LIN {X 0,Y 407.293,Z 572.545,A -85,B 0,C 180,E1 -11318.769,E2 -11318.769} C_VEL
LIN {X 0,Y 407.261,Z 605.136,A -85,B 0,C 180,E1 -11319.46,E2 -11319.46} C_VEL
LIN {X 0,Y 407.213,Z 619.891,A -85,B 0,C 180,E1 -11319.972,E2 -11319.972} C_VEL
LIN {X 0,Y 406.821,Z 633.745,A -85,B 0,C 180,E1 -11320.641,E2 -11320.641} C_VEL
LIN {X 0,Y 406.274,Z 646.742,A -85,B 0,C 180,E1 -11321.466,E2 -11321.466} C_VEL
LIN {X 0,Y 405.576,Z 659.147,A -85,B 0,C 180,E1 -11322.444,E2 -11322.444} C_VEL
LIN {X 0,Y 404.643,Z 671.423,A -85,B 0,C 180,E1 -11323.636,E2 -11323.636} C_VEL
LIN {X 0,Y 403.725,Z 681.881,A -85,B 0,C 180,E1 -11324.863,E2 -11324.863} C_VEL
LIN {X 0,Y 402.584,Z 692.537,A -85,B 0,C 180,E1 -11326.368,E2 -11326.368} C_VEL
LIN {X 0,Y 401.584,Z 701.412,A -85,B 0,C 180,E1 -11327.877,E2 -11327.877} C_VEL
LIN {X 0,Y 400.622,Z 709.855,A -85,B 0,C 180,E1 -11329.61,E2 -11329.61} C_VEL
LIN {X 0,Y 399.757,Z 716.985,A -85,B 0,C 180,E1 -11331.405,E2 -11331.405} C_VEL
LIN {X 0,Y 398.956,Z 721.911,A -85,B 0,C 180,E1 -11332.916,E2 -11332.916} C_VEL
LIN {X 0,Y 398.421,Z 727.092,A -85,B 0,C 180,E1 -11334.94,E2 -11334.94} C_VEL
LIN {X 0,Y 397.856,Z 730.905,A -85,B 0,C 180,E1 -11336.962,E2 -11336.962} C_VEL
LIN {X 0,Y 397.512,Z 733.428,A -85,B 0,C 180,E1 -11338.987,E2 -11338.987} C_VEL
LIN {X 0,Y 397.294,Z 734.718,A -85,B 0,C 180,E1 -11341.013,E2 -11341.013} C_VEL
LIN {X 0,Y 397.207,Z 734.793,A -85,B 0,C 180,E1 -11343.042,E2 -11343.042} C_VEL
LIN {X 0,Y 397.117,Z 733.67,A -85,B 0,C 180,E1 -11345.076,E2 -11345.076} C_VEL
LIN {X 0,Y 397.307,Z 731.92,A -85,B 0,C 180,E1 -11346.634,E2 -11346.634} C_VEL
LIN {X 0,Y 397.376,Z 729.649,A -85,B 0,C 180,E1 -11348.133,E2 -11348.133} C_VEL
LIN {X 0,Y 397.643,Z 725.336,A -85,B 0,C 180,E1 -11350.18,E2 -11350.18} C_VEL
LIN {X 0,Y 397.959,Z 719.588,A -85,B 0,C 180,E1 -11352.234,E2 -11352.234} C_VEL
LIN {X 0,Y 398.554,Z 712.207,A -85,B 0,C 180,E1 -11354.292,E2 -11354.292} C_VEL
LIN {X 0,Y 399.245,Z 704.203,A -85,B 0,C 180,E1 -11356.096,E2 -11356.096} C_VEL
LIN {X 0,Y 400.049,Z 694.472,A -85,B 0,C 180,E1 -11357.904,E2 -11357.904} C_VEL
LIN {X 0,Y 400.824,Z 684.417,A -85,B 0,C 180,E1 -11359.459,E2 -11359.459} C_VEL
LIN {X 0,Y 401.695,Z 673.415,A -85,B 0,C 180,E1 -11360.884,E2 -11360.884} C_VEL
LIN {X 0,Y 402.54,Z 661.884,A -85,B 0,C 180,E1 -11362.136,E2 -11362.136} C_VEL
LIN {X 0,Y 403.272,Z 649.96,A -85,B 0,C 180,E1 -11363.222,E2 -11363.222} C_VEL
LIN {X 0,Y 404.01,Z 635.883,A -85,B 0,C 180,E1 -11364.265,E2 -11364.265} C_VEL
LIN {X 0,Y 404.662,Z 621.146,A -85,B 0,C 180,E1 -11365.12,E2 -11365.12} C_VEL
LIN {X 0,Y 405.075,Z 605.669,A -85,B 0,C 180,E1 -11365.793,E2 -11365.793} C_VEL
LIN {X 0,Y 405.206,Z 590.616,A -85,B 0,C 180,E1 -11366.244,E2 -11366.244} C_VEL
LIN {X 0,Y 405.225,Z 572.67,A -85,B 0,C 180,E1 -11366.637,E2 -11366.637} C_VEL
LIN {X 0,Y 397.184,Z 551.01,A -85,B 0,C 180,E1 -11367.501,E2 -11367.501} C_VEL
LIN {X 0,Y 397.08,Z 551.019,A -85,B 0,C 180,E1 -11370.882,E2 -11370.882} C_VEL
LIN {X 0,Y 397.126,Z 551.016,A -85,B 0,C 180,E1 -11374.493,E2 -11374.493} C_VEL
LIN {X 0,Y 397.103,Z 551.022,A -85,B 0,C 180,E1 -11378.274,E2 -11378.274} C_VEL
LIN {X 0,Y 397.089,Z 551.018,A -85,B 0,C 180,E1 -11380.908,E2 -11380.908} C_VEL
LIN {X 0,Y 397.101,Z 551.017,A -85,B 0,C 180,E1 -11383.648,E2 -11383.648} C_VEL
LIN {X 0,Y 397.102,Z 551.021,A -85,B 0,C 180,E1 -11386.52,E2 -11386.52} C_VEL
LIN {X 0,Y 397.115,Z 551.022,A -85,B 0,C 180,E1 -11390.422,E2 -11390.422} C_VEL
LIN {X 0,Y 397.108,Z 551.02,A -85,B 0,C 180,E1 -11394.265,E2 -11394.265} C_VEL
LIN {X 0,Y 397.114,Z 551.019,A -85,B 0,C 180,E1 -11396.726,E2 -11396.726} C_VEL
LIN {X 0,Y 397.124,Z 551.017,A -85,B 0,C 180,E1 -11400.295,E2 -11400.295} C_VEL
LIN {X 0,Y 397.193,Z 551.012,A -85,B 0,C 180,E1 -11402.609,E2 -11402.609} C_VEL
LIN {X 0,Y 397.132,Z 551.013,A -85,B 0,C 180,E1 -11405.981,E2 -11405.981} C_VEL
LIN {X 0,Y 397.137,Z 551.011,A -85,B 0,C 180,E1 -11409.704,E2 -11409.704} C_VEL
LIN {X 0,Y 397.18,Z 551.014,A -85,B 0,C 180,E1 -11412.844,E2 -11412.844} C_VEL
LIN {X 0,Y 397.225,Z 551.005,A -85,B 0,C 180,E1 -11416.678,E2 -11416.678} C_VEL
LIN {X 0,Y 397.217,Z 551.002,A -85,B 0,C 180,E1 -11419.808,E2 -11419.808} C_VEL
LIN {X 0,Y 397.362,Z 550.989,A -85,B 0,C 180,E1 -11422.888,E2 -11422.888} C_VEL
LIN {X 0,Y 397.254,Z 551.003,A -85,B 0,C 180,E1 -11424.925,E2 -11424.925} C_VEL
LIN {X 0,Y 397.45,Z 550.973,A -85,B 0,C 180,E1 -11427.973,E2 -11427.973} C_VEL
LIN {X 0,Y 397.579,Z 550.957,A -85,B 0,C 180,E1 -11429.999,E2 -11429.999} C_VEL
LIN {X 0,Y 397.38,Z 550.987,A -85,B 0,C 180,E1 -11433.041,E2 -11433.041} C_VEL
LIN {X 0,Y 397.357,Z 550.989,A -85,B 0,C 180,E1 -11437.111,E2 -11437.111} C_VEL
LIN {X 0,Y 397.22,Z 551.001,A -85,B 0,C 180,E1 -11440.19,E2 -11440.19} C_VEL
LIN {X 0,Y 397.223,Z 551.008,A -85,B 0,C 180,E1 -11443.32,E2 -11443.32} C_VEL
LIN {X 0,Y 397.165,Z 551.009,A -85,B 0,C 180,E1 -11446.89,E2 -11446.89} C_VEL
LIN {X 0,Y 396.521,Z 551.096,A -85,B 0,C 180,E1 -11447.737,E2 -11447.737} C_VEL
LIN {X 0,Y 393.659,Z 551.454,A -85,B 0,C 180,E1 -11449.111,E2 -11449.111} C_VEL
LIN {X 0,Y 391.208,Z 551.757,A -85,B 0,C 180,E1 -11450.222,E2 -11450.222} C_VEL
LIN {X 0,Y 390.138,Z 551.886,A -85,B 0,C 180,E1 -11451.081,E2 -11451.081} C_VEL
LIN {X 0,Y 390.042,Z 551.896,A -85,B 0,C 180,E1 -11451.373,E2 -11451.373} C_VEL
LIN {X 0,Y 390.076,Z 551.891,A -85,B 0,C 180,E1 -11454.48,E2 -11454.48} C_VEL
LIN {X 0,Y 390.111,Z 551.89,A -85,B 0,C 180,E1 -11458.025,E2 -11458.025} C_VEL
LIN {X 0,Y 390.045,Z 551.9,A -85,B 0,C 180,E1 -11461.502,E2 -11461.502} C_VEL
LIN {X 0,Y 390.081,Z 551.892,A -85,B 0,C 180,E1 -11465.206,E2 -11465.206} C_VEL
LIN {X 0,Y 390.089,Z 551.89,A -85,B 0,C 180,E1 -11469.091,E2 -11469.091} C_VEL
LIN {X 0,Y 390.075,Z 551.893,A -85,B 0,C 180,E1 -11472.38,E2 -11472.38} C_VEL
LIN {X 0,Y 390.1,Z 551.894,A -85,B 0,C 180,E1 -11476.106,E2 -11476.106} C_VEL
LIN {X 0,Y 390.078,Z 551.891,A -85,B 0,C 180,E1 -11479.174,E2 -11479.174} C_VEL
LIN {X 0,Y 390.042,Z 551.899,A -85,B 0,C 180,E1 -11482.448,E2 -11482.448} C_VEL
LIN {X 0,Y 390.103,Z 551.888,A -85,B 0,C 180,E1 -11484.796,E2 -11484.796} C_VEL
LIN {X 0,Y 394.039,Z 562.764,A -85,B 0,C 180,E1 -11485.247,E2 -11485.247} C_VEL
LIN {X 0,Y 397.384,Z 571.668,A -85,B 0,C 180,E1 -11485.586,E2 -11485.586} C_VEL
LIN {X 0,Y 396.866,Z 611.928,A -85,B 0,C 180,E1 -11486.443,E2 -11486.443} C_VEL
LIN {X 0,Y 396.685,Z 626.411,A -85,B 0,C 180,E1 -11486.952,E2 -11486.952} C_VEL
LIN {X 0,Y 396.218,Z 639.939,A -85,B 0,C 180,E1 -11487.626,E2 -11487.626} C_VEL
LIN {X 0,Y 395.593,Z 653.284,A -85,B 0,C 180,E1 -11488.511,E2 -11488.511} C_VEL
LIN {X 0,Y 394.939,Z 665.36,A -85,B 0,C 180,E1 -11489.526,E2 -11489.526} C_VEL
LIN {X 0,Y 394.119,Z 677.299,A -85,B 0,C 180,E1 -11490.759,E2 -11490.759} C_VEL
LIN {X 0,Y 393.25,Z 688.447,A -85,B 0,C 180,E1 -11492.168,E2 -11492.168} C_VEL
LIN {X 0,Y 392.574,Z 698.027,A -85,B 0,C 180,E1 -11493.647,E2 -11493.647} C_VEL
LIN {X 0,Y 391.781,Z 707.081,A -85,B 0,C 180,E1 -11495.351,E2 -11495.351} C_VEL
LIN {X 0,Y 391.137,Z 715.317,A -85,B 0,C 180,E1 -11497.275,E2 -11497.275} C_VEL
LIN {X 0,Y 390.706,Z 720.929,A -85,B 0,C 180,E1 -11498.915,E2 -11498.915} C_VEL
LIN {X 0,Y 390.388,Z 725.399,A -85,B 0,C 180,E1 -11500.547,E2 -11500.547} C_VEL
LIN {X 0,Y 390.137,Z 728.855,A -85,B 0,C 180,E1 -11502.168,E2 -11502.168} C_VEL
LIN {X 0,Y 389.957,Z 732.027,A -85,B 0,C 180,E1 -11504.316,E2 -11504.316} C_VEL
LIN {X 0,Y 389.954,Z 733.693,A -85,B 0,C 180,E1 -11506.45,E2 -11506.45} C_VEL
LIN {X 0,Y 390.064,Z 733.846,A -85,B 0,C 180,E1 -11508.569,E2 -11508.569} C_VEL
LIN {X 0,Y 390.276,Z 732.579,A -85,B 0,C 180,E1 -11510.673,E2 -11510.673} C_VEL
LIN {X 0,Y 390.669,Z 729.882,A -85,B 0,C 180,E1 -11512.766,E2 -11512.766} C_VEL
LIN {X 0,Y 391.058,Z 726.833,A -85,B 0,C 180,E1 -11514.328,E2 -11514.328} C_VEL
LIN {X 0,Y 391.699,Z 721.406,A -85,B 0,C 180,E1 -11516.4,E2 -11516.4} C_VEL
LIN {X 0,Y 392.504,Z 715.104,A -85,B 0,C 180,E1 -11518.205,E2 -11518.205} C_VEL
LIN {X 0,Y 393.31,Z 707.265,A -85,B 0,C 180,E1 -11520,E2 -11520} C_VEL
LIN {X 0,Y 394.268,Z 699.146,A -85,B 0,C 180,E1 -11521.5,E2 -11521.5} C_VEL
LIN {X 0,Y 395.266,Z 688.896,A -85,B 0,C 180,E1 -11523.058,E2 -11523.058} C_VEL
LIN {X 0,Y 396.207,Z 678.627,A -85,B 0,C 180,E1 -11524.324,E2 -11524.324} C_VEL
LIN {X 0,Y 397.067,Z 667.326,A -85,B 0,C 180,E1 -11525.46,E2 -11525.46} C_VEL
LIN {X 0,Y 397.871,Z 654.762,A -85,B 0,C 180,E1 -11526.466,E2 -11526.466} C_VEL
LIN {X 0,Y 398.394,Z 641.791,A -85,B 0,C 180,E1 -11527.285,E2 -11527.285} C_VEL
LIN {X 0,Y 398.774,Z 628.326,A -85,B 0,C 180,E1 -11527.915,E2 -11527.915} C_VEL
LIN {X 0,Y 398.873,Z 613.965,A -85,B 0,C 180,E1 -11528.362,E2 -11528.362} C_VEL
LIN {X 0,Y 399.365,Z 578.05,A -85,B 0,C 180,E1 -11529.113,E2 -11529.113} C_VEL
LIN {X 0,Y 399.421,Z 572.286,A -85,B 0,C 180,E1 -11529.237,E2 -11529.237} C_VEL
LIN {X 0,Y 395.215,Z 562.731,A -85,B 0,C 180,E1 -11529.765,E2 -11529.765} C_VEL
LIN {X 0,Y 390.328,Z 552.675,A -85,B 0,C 180,E1 -11530.4,E2 -11530.4} C_VEL
LIN {X 0,Y 390.164,Z 551.886,A -85,B 0,C 180,E1 -11530.443,E2 -11530.443} C_VEL
LIN {X 0,Y 390.166,Z 551.889,A -85,B 0,C 180,E1 -11533.543,E2 -11533.543} C_VEL
LIN {X 0,Y 390.145,Z 551.893,A -85,B 0,C 180,E1 -11537.308,E2 -11537.308} C_VEL
LIN {X 0,Y 390.084,Z 551.895,A -85,B 0,C 180,E1 -11540.471,E2 -11540.471} C_VEL
LIN {X 0,Y 390.086,Z 551.893,A -85,B 0,C 180,E1 -11543.351,E2 -11543.351} C_VEL
LIN {X 0,Y 390.111,Z 551.888,A -85,B 0,C 180,E1 -11546.769,E2 -11546.769} C_VEL
LIN {X 0,Y 390.042,Z 551.891,A -85,B 0,C 180,E1 -11550.3,E2 -11550.3} C_VEL
LIN {X 0,Y 390.066,Z 551.888,A -85,B 0,C 180,E1 -11554.025,E2 -11554.025} C_VEL
LIN {X 0,Y 390.044,Z 551.896,A -85,B 0,C 180,E1 -11557.552,E2 -11557.552} C_VEL
LIN {X 0,Y 390.056,Z 551.897,A -85,B 0,C 180,E1 -11560.822,E2 -11560.822} C_VEL
LIN {X 0,Y 390.056,Z 551.895,A -85,B 0,C 180,E1 -11563.887,E2 -11563.887} C_VEL
LIN {X 0,Y 390.056,Z 551.897,A -85,B 0,C 180,E1 -11566.79,E2 -11566.79} C_VEL
LIN {X 0,Y 390.055,Z 551.894,A -85,B 0,C 180,E1 -11569.561,E2 -11569.561} C_VEL
LIN {X 0,Y 390.099,Z 552.016,A -85,B 0,C 180,E1 -11572.492,E2 -11572.492} C_VEL
LIN {X 0,Y 393.227,Z 566.767,A -85,B 0,C 180,E1 -11576.067,E2 -11576.067} C_VEL
LIN {X 0,Y 394.741,Z 573.819,A -85,B 0,C 180,E1 -11577.716,E2 -11577.716} C_VEL
LIN {X 0,Y 394.326,Z 580.533,A -85,B 0,C 180,E1 -11579.177,E2 -11579.177} C_VEL
LIN {X 0,Y 392.928,Z 596.517,A -85,B 0,C 180,E1 -11582.577,E2 -11582.577} C_VEL
LIN {X 0,Y 391.812,Z 612.738,A -85,B 0,C 180,E1 -11585.98,E2 -11585.98} C_VEL
LIN {X 0,Y 391.001,Z 625.883,A -85,B 0,C 180,E1 -11588.718,E2 -11588.718} C_VEL
LIN {X 0,Y 395.028,Z 659.806,A -85,B 0,C 180,E1 -11589.871,E2 -11589.871} C_VEL
LIN {X 0,Y 396.868,Z 676.408,A -85,B 0,C 180,E1 -11590.386,E2 -11590.386} C_VEL
LIN {X 0,Y 395.687,Z 721.414,A -85,B 0,C 180,E1 -11591.456,E2 -11591.456} C_VEL
LIN {X 0,Y 395.233,Z 737.692,A -85,B 0,C 180,E1 -11591.87,E2 -11591.87} C_VEL
LIN {X 0,Y 394.335,Z 755.406,A -85,B 0,C 180,E1 -11592.565,E2 -11592.565} C_VEL
LIN {X 0,Y 393.397,Z 767.999,A -85,B 0,C 180,E1 -11593.258,E2 -11593.258} C_VEL
LIN {X 0,Y 392.457,Z 780.282,A -85,B 0,C 180,E1 -11594.152,E2 -11594.152} C_VEL
LIN {X 0,Y 391.614,Z 791.534,A -85,B 0,C 180,E1 -11595.184,E2 -11595.184} C_VEL
LIN {X 0,Y 390.704,Z 802.918,A -85,B 0,C 180,E1 -11596.477,E2 -11596.477} C_VEL
LIN {X 0,Y 390.235,Z 810.509,A -85,B 0,C 180,E1 -11597.52,E2 -11597.52} C_VEL
LIN {X 0,Y 389.681,Z 819.933,A -85,B 0,C 180,E1 -11599.085,E2 -11599.085} C_VEL
LIN {X 0,Y 389.375,Z 827.561,A -85,B 0,C 180,E1 -11600.652,E2 -11600.652} C_VEL
LIN {X 0,Y 389.276,Z 833.694,A -85,B 0,C 180,E1 -11602.219,E2 -11602.219} C_VEL
LIN {X 0,Y 389.294,Z 838.509,A -85,B 0,C 180,E1 -11603.782,E2 -11603.782} C_VEL
LIN {X 0,Y 389.459,Z 842.149,A -85,B 0,C 180,E1 -11605.343,E2 -11605.343} C_VEL
LIN {X 0,Y 389.48,Z 844.657,A -85,B 0,C 180,E1 -11606.897,E2 -11606.897} C_VEL
LIN {X 0,Y 389.498,Z 845.766,A -85,B 0,C 180,E1 -11607.933,E2 -11607.933} C_VEL
LIN {X 0,Y 389.534,Z 846.387,A -85,B 0,C 180,E1 -11608.967,E2 -11608.967} C_VEL
LIN {X 0,Y 389.775,Z 846.585,A -85,B 0,C 180,E1 -11610.001,E2 -11610.001} C_VEL
LIN {X 0,Y 389.546,Z 846.274,A -85,B 0,C 180,E1 -11611.034,E2 -11611.034} C_VEL
LIN {X 0,Y 389.515,Z 845.556,A -85,B 0,C 180,E1 -11612.069,E2 -11612.069} C_VEL
LIN {X 0,Y 389.503,Z 844.358,A -85,B 0,C 180,E1 -11613.104,E2 -11613.104} C_VEL
LIN {X 0,Y 389.484,Z 841.719,A -85,B 0,C 180,E1 -11614.658,E2 -11614.658} C_VEL
LIN {X 0,Y 389.366,Z 837.972,A -85,B 0,C 180,E1 -11616.218,E2 -11616.218} C_VEL
LIN {X 0,Y 389.287,Z 833.061,A -85,B 0,C 180,E1 -11617.782,E2 -11617.782} C_VEL
LIN {X 0,Y 389.366,Z 826.882,A -85,B 0,C 180,E1 -11619.35,E2 -11619.35} C_VEL
LIN {X 0,Y 389.632,Z 819.251,A -85,B 0,C 180,E1 -11620.918,E2 -11620.918} C_VEL
LIN {X 0,Y 390.169,Z 809.947,A -85,B 0,C 180,E1 -11622.484,E2 -11622.484} C_VEL
LIN {X 0,Y 390.689,Z 800.971,A -85,B 0,C 180,E1 -11623.736,E2 -11623.736} C_VEL
LIN {X 0,Y 391.437,Z 791.747,A -85,B 0,C 180,E1 -11624.824,E2 -11624.824} C_VEL
LIN {X 0,Y 392.587,Z 779.948,A -85,B 0,C 180,E1 -11625.977,E2 -11625.977} C_VEL
LIN {X 0,Y 393.759,Z 766.955,A -85,B 0,C 180,E1 -11626.994,E2 -11626.994} C_VEL
LIN {X 0,Y 395.052,Z 752.51,A -85,B 0,C 180,E1 -11627.872,E2 -11627.872} C_VEL
LIN {X 0,Y 396.1,Z 737.875,A -85,B 0,C 180,E1 -11628.525,E2 -11628.525} C_VEL
LIN {X 0,Y 396.711,Z 722.721,A -85,B 0,C 180,E1 -11628.998,E2 -11628.998} C_VEL
LIN {X 0,Y 398.047,Z 674.809,A -85,B 0,C 180,E1 -11630.157,E2 -11630.157} C_VEL
LIN {X 0,Y 396.794,Z 652.456,A -85,B 0,C 180,E1 -11630.859,E2 -11630.859} C_VEL
LIN {X 0,Y 395.347,Z 634.248,A -85,B 0,C 180,E1 -11631.486,E2 -11631.486} C_VEL
LIN {X 0,Y 392.774,Z 614.765,A -85,B 0,C 180,E1 -11632.274,E2 -11632.274} C_VEL
LIN {X 0,Y 390.428,Z 600.878,A -85,B 0,C 180,E1 -11632.909,E2 -11632.909} C_VEL
LIN {X 0,Y 390.923,Z 582.654,A -85,B 0,C 180,E1 -11636.492,E2 -11636.492} C_VEL
LIN {X 0,Y 391.662,Z 564.675,A -85,B 0,C 180,E1 -11640.162,E2 -11640.162} C_VEL
LIN {X 0,Y 391.627,Z 560.084,A -85,B 0,C 180,E1 -11641.133,E2 -11641.133} C_VEL
LIN {X 0,Y 390.122,Z 551.895,A -85,B 0,C 180,E1 -11643.022,E2 -11643.022} C_VEL
LIN {X 0,Y 390.062,Z 551.896,A -85,B 0,C 180,E1 -11646.483,E2 -11646.483} C_VEL
LIN {X 0,Y 390.074,Z 551.896,A -85,B 0,C 180,E1 -11649.218,E2 -11649.218} C_VEL
LIN {X 0,Y 390.046,Z 551.897,A -85,B 0,C 180,E1 -11652.374,E2 -11652.374} C_VEL
LIN {X 0,Y 390.049,Z 551.899,A -85,B 0,C 180,E1 -11655.354,E2 -11655.354} C_VEL
LIN {X 0,Y 390.036,Z 551.899,A -85,B 0,C 180,E1 -11658.187,E2 -11658.187} C_VEL
LIN {X 0,Y 390.095,Z 551.893,A -85,B 0,C 180,E1 -11660.908,E2 -11660.908} C_VEL
LIN {X 0,Y 390.089,Z 551.894,A -85,B 0,C 180,E1 -11664.793,E2 -11664.793} C_VEL
LIN {X 0,Y 390.028,Z 551.902,A -85,B 0,C 180,E1 -11668.496,E2 -11668.496} C_VEL
LIN {X 0,Y 390.122,Z 551.893,A -85,B 0,C 180,E1 -11672.07,E2 -11672.07} C_VEL
LIN {X 0,Y 390.085,Z 551.897,A -85,B 0,C 180,E1 -11675.519,E2 -11675.519} C_VEL
LIN {X 0,Y 390.101,Z 551.896,A -85,B 0,C 180,E1 -11676.816,E2 -11676.816} C_VEL
LIN {X 0,Y 391.195,Z 554.921,A -85,B 0,C 180,E1 -11677.009,E2 -11677.009} C_VEL
LIN {X 0,Y 392.415,Z 556.899,A -85,B 0,C 180,E1 -11677.171,E2 -11677.171} C_VEL
LIN {X 0,Y 398.945,Z 569.682,A -85,B 0,C 180,E1 -11678.037,E2 -11678.037} C_VEL
LIN {X 0,Y 401.155,Z 575.073,A -85,B 0,C 180,E1 -11678.339,E2 -11678.339} C_VEL
LIN {X 0,Y 400.947,Z 604.204,A -85,B 0,C 180,E1 -11678.97,E2 -11678.97} C_VEL
LIN {X 0,Y 400.936,Z 619.083,A -85,B 0,C 180,E1 -11679.455,E2 -11679.455} C_VEL
LIN {X 0,Y 400.607,Z 633.41,A -85,B 0,C 180,E1 -11680.129,E2 -11680.129} C_VEL
LIN {X 0,Y 400.068,Z 645.882,A -85,B 0,C 180,E1 -11680.902,E2 -11680.902} C_VEL
LIN {X 0,Y 399.3,Z 658.587,A -85,B 0,C 180,E1 -11681.888,E2 -11681.888} C_VEL
LIN {X 0,Y 398.307,Z 670.965,A -85,B 0,C 180,E1 -11683.074,E2 -11683.074} C_VEL
LIN {X 0,Y 397.281,Z 681.934,A -85,B 0,C 180,E1 -11684.349,E2 -11684.349} C_VEL
LIN {X 0,Y 396.126,Z 692.845,A -85,B 0,C 180,E1 -11685.88,E2 -11685.88} C_VEL
LIN {X 0,Y 395.038,Z 701.861,A -85,B 0,C 180,E1 -11687.412,E2 -11687.412} C_VEL
LIN {X 0,Y 393.94,Z 710.759,A -85,B 0,C 180,E1 -11689.249,E2 -11689.249} C_VEL
LIN {X 0,Y 392.915,Z 718.55,A -85,B 0,C 180,E1 -11691.255,E2 -11691.255} C_VEL
LIN {X 0,Y 392.081,Z 723.432,A -85,B 0,C 180,E1 -11692.791,E2 -11692.791} C_VEL
LIN {X 0,Y 391.505,Z 728.532,A -85,B 0,C 180,E1 -11694.85,E2 -11694.85} C_VEL
LIN {X 0,Y 390.91,Z 732.26,A -85,B 0,C 180,E1 -11696.908,E2 -11696.908} C_VEL
LIN {X 0,Y 390.543,Z 734.677,A -85,B 0,C 180,E1 -11698.968,E2 -11698.968} C_VEL
LIN {X 0,Y 390.297,Z 735.864,A -85,B 0,C 180,E1 -11701.031,E2 -11701.031} C_VEL
LIN {X 0,Y 390.186,Z 735.839,A -85,B 0,C 180,E1 -11703.097,E2 -11703.097} C_VEL
LIN {X 0,Y 390.103,Z 734.615,A -85,B 0,C 180,E1 -11705.168,E2 -11705.168} C_VEL
LIN {X 0,Y 390.296,Z 732.949,A -85,B 0,C 180,E1 -11706.629,E2 -11706.629} C_VEL
LIN {X 0,Y 390.432,Z 729.467,A -85,B 0,C 180,E1 -11708.801,E2 -11708.801} C_VEL
LIN {X 0,Y 390.726,Z 724.683,A -85,B 0,C 180,E1 -11710.886,E2 -11710.886} C_VEL
LIN {X 0,Y 391.151,Z 718.411,A -85,B 0,C 180,E1 -11712.978,E2 -11712.978} C_VEL
LIN {X 0,Y 391.707,Z 711.512,A -85,B 0,C 180,E1 -11714.813,E2 -11714.813} C_VEL
LIN {X 0,Y 392.45,Z 703.105,A -85,B 0,C 180,E1 -11716.65,E2 -11716.65} C_VEL
LIN {X 0,Y 393.291,Z 693.473,A -85,B 0,C 180,E1 -11718.392,E2 -11718.392} C_VEL
LIN {X 0,Y 394.156,Z 682.262,A -85,B 0,C 180,E1 -11720.074,E2 -11720.074} C_VEL
LIN {X 0,Y 395.033,Z 670.588,A -85,B 0,C 180,E1 -11721.526,E2 -11721.526} C_VEL
LIN {X 0,Y 395.954,Z 657.881,A -85,B 0,C 180,E1 -11722.835,E2 -11722.835} C_VEL
LIN {X 0,Y 396.783,Z 645.309,A -85,B 0,C 180,E1 -11723.901,E2 -11723.901} C_VEL
LIN {X 0,Y 397.433,Z 631.83,A -85,B 0,C 180,E1 -11724.833,E2 -11724.833} C_VEL
LIN {X 0,Y 398.055,Z 616.78,A -85,B 0,C 180,E1 -11725.637,E2 -11725.637} C_VEL
LIN {X 0,Y 398.335,Z 601.5,A -85,B 0,C 180,E1 -11726.238,E2 -11726.238} C_VEL
LIN {X 0,Y 398.481,Z 585.129,A -85,B 0,C 180,E1 -11726.663,E2 -11726.663} C_VEL
LIN {X 0,Y 398.498,Z 574.488,A -85,B 0,C 180,E1 -11726.896,E2 -11726.896} C_VEL
LIN {X 0,Y 390.113,Z 551.893,A -85,B 0,C 180,E1 -11727.836,E2 -11727.836} C_VEL
LIN {X 0,Y 390.025,Z 551.899,A -85,B 0,C 180,E1 -11731.504,E2 -11731.504} C_VEL
LIN {X 0,Y 390.086,Z 551.89,A -85,B 0,C 180,E1 -11735.206,E2 -11735.206} C_VEL
LIN {X 0,Y 390.07,Z 551.892,A -85,B 0,C 180,E1 -11739.218,E2 -11739.218} C_VEL
LIN {X 0,Y 390.043,Z 551.901,A -85,B 0,C 180,E1 -11742.373,E2 -11742.373} C_VEL
LIN {X 0,Y 390.044,Z 551.895,A -85,B 0,C 180,E1 -11745.354,E2 -11745.354} C_VEL
LIN {X 0,Y 390.031,Z 551.902,A -85,B 0,C 180,E1 -11748.186,E2 -11748.186} C_VEL
LIN {X 0,Y 390.092,Z 551.891,A -85,B 0,C 180,E1 -11750.907,E2 -11750.907} C_VEL
LIN {X 0,Y 390.085,Z 551.894,A -85,B 0,C 180,E1 -11754.793,E2 -11754.793} C_VEL
LIN {X 0,Y 390.023,Z 551.904,A -85,B 0,C 180,E1 -11758.495,E2 -11758.495} C_VEL
LIN {X 0,Y 390.116,Z 551.888,A -85,B 0,C 180,E1 -11762.069,E2 -11762.069} C_VEL
LIN {X 0,Y 390.079,Z 551.891,A -85,B 0,C 180,E1 -11765.519,E2 -11765.519} C_VEL
LIN {X 0,Y 390.055,Z 551.9,A -85,B 0,C 180,E1 -11768.877,E2 -11768.877} C_VEL
LIN {X 0,Y 390.127,Z 551.886,A -85,B 0,C 180,E1 -11772.166,E2 -11772.166} C_VEL
LIN {X 0,Y 390.143,Z 551.884,A -85,B 0,C 180,E1 -11775.392,E2 -11775.392} C_VEL
LIN {X 0,Y 390.147,Z 551.885,A -85,B 0,C 180,E1 -11778.571,E2 -11778.571} C_VEL
LIN {X 0,Y 390.342,Z 551.858,A -85,B 0,C 180,E1 -11781.992,E2 -11781.992} C_VEL
LIN {X 0,Y 390.226,Z 551.877,A -85,B 0,C 180,E1 -11784.833,E2 -11784.833} C_VEL
LIN {X 0,Y 390.418,Z 551.849,A -85,B 0,C 180,E1 -11787.936,E2 -11787.936} C_VEL
LIN {X 0,Y 390.548,Z 551.832,A -85,B 0,C 180,E1 -11789.999,E2 -11789.999} C_VEL
LIN {X 0,Y 390.314,Z 551.868,A -85,B 0,C 180,E1 -11793.096,E2 -11793.096} C_VEL
LIN {X 0,Y 390.324,Z 551.86,A -85,B 0,C 180,E1 -11796.201,E2 -11796.201} C_VEL
LIN {X 0,Y 390.312,Z 551.862,A -85,B 0,C 180,E1 -11798.282,E2 -11798.282} C_VEL
LIN {X 0,Y 390.176,Z 551.879,A -85,B 0,C 180,E1 -11802.482,E2 -11802.482} C_VEL
LIN {X 0,Y 390.137,Z 551.888,A -85,B 0,C 180,E1 -11805.676,E2 -11805.676} C_VEL
LIN {X 0,Y 390.102,Z 551.889,A -85,B 0,C 180,E1 -11808.922,E2 -11808.922} C_VEL
LIN {X 0,Y 390.042,Z 551.896,A -85,B 0,C 180,E1 -11811.373,E2 -11811.373} C_VEL
LIN {X 0,Y 389.349,Z 551.984,A -85,B 0,C 180,E1 -11812.234,E2 -11812.234} C_VEL
LIN {X 0,Y 386.488,Z 552.345,A -85,B 0,C 180,E1 -11813.635,E2 -11813.635} C_VEL
LIN {X 0,Y 384.11,Z 552.636,A -85,B 0,C 180,E1 -11814.767,E2 -11814.767} C_VEL
LIN {X 0,Y 383.131,Z 552.763,A -85,B 0,C 180,E1 -11815.643,E2 -11815.643} C_VEL
LIN {X 0,Y 383.072,Z 552.766,A -85,B 0,C 180,E1 -11815.939,E2 -11815.939} C_VEL
LIN {X 0,Y 383.047,Z 552.767,A -85,B 0,C 180,E1 -11818.491,E2 -11818.491} C_VEL
LIN {X 0,Y 383.032,Z 552.771,A -85,B 0,C 180,E1 -11822.147,E2 -11822.147} C_VEL
LIN {X 0,Y 383.022,Z 552.775,A -85,B 0,C 180,E1 -11825.955,E2 -11825.955} C_VEL
LIN {X 0,Y 383.016,Z 552.774,A -85,B 0,C 180,E1 -11829.587,E2 -11829.587} C_VEL
LIN {X 0,Y 383.027,Z 552.769,A -85,B 0,C 180,E1 -11832.783,E2 -11832.783} C_VEL
LIN {X 0,Y 383.036,Z 552.773,A -85,B 0,C 180,E1 -11835.796,E2 -11835.796} C_VEL
LIN {X 0,Y 383.039,Z 552.768,A -85,B 0,C 180,E1 -11838.786,E2 -11838.786} C_VEL
LIN {X 0,Y 382.998,Z 552.78,A -85,B 0,C 180,E1 -11842.095,E2 -11842.095} C_VEL
LIN {X 0,Y 383.04,Z 552.771,A -85,B 0,C 180,E1 -11844.498,E2 -11844.498} C_VEL
LIN {X 0,Y 390.638,Z 573.589,A -85,B 0,C 180,E1 -11845.326,E2 -11845.326} C_VEL
LIN {X 0,Y 390.04,Z 612.522,A -85,B 0,C 180,E1 -11846.172,E2 -11846.172} C_VEL
LIN {X 0,Y 389.854,Z 626.985,A -85,B 0,C 180,E1 -11846.684,E2 -11846.684} C_VEL
LIN {X 0,Y 389.376,Z 640.665,A -85,B 0,C 180,E1 -11847.371,E2 -11847.371} C_VEL
LIN {X 0,Y 388.731,Z 654.215,A -85,B 0,C 180,E1 -11848.282,E2 -11848.282} C_VEL
LIN {X 0,Y 387.991,Z 666.942,A -85,B 0,C 180,E1 -11849.373,E2 -11849.373} C_VEL
LIN {X 0,Y 387.139,Z 678.982,A -85,B 0,C 180,E1 -11850.65,E2 -11850.65} C_VEL
LIN {X 0,Y 386.289,Z 689.883,A -85,B 0,C 180,E1 -11852.064,E2 -11852.064} C_VEL
LIN {X 0,Y 385.558,Z 699.524,A -85,B 0,C 180,E1 -11853.595,E2 -11853.595} C_VEL
LIN {X 0,Y 384.848,Z 707.744,A -85,B 0,C 180,E1 -11855.165,E2 -11855.165} C_VEL
LIN {X 0,Y 384.267,Z 714.99,A -85,B 0,C 180,E1 -11856.845,E2 -11856.845} C_VEL
LIN {X 0,Y 383.765,Z 720.881,A -85,B 0,C 180,E1 -11858.515,E2 -11858.515} C_VEL
LIN {X 0,Y 383.436,Z 725.607,A -85,B 0,C 180,E1 -11860.179,E2 -11860.179} C_VEL
LIN {X 0,Y 383.154,Z 729.294,A -85,B 0,C 180,E1 -11861.831,E2 -11861.831} C_VEL
LIN {X 0,Y 382.937,Z 732.689,A -85,B 0,C 180,E1 -11864.021,E2 -11864.021} C_VEL
LIN {X 0,Y 382.922,Z 734.572,A -85,B 0,C 180,E1 -11866.197,E2 -11866.197} C_VEL
LIN {X 0,Y 383.06,Z 734.995,A -85,B 0,C 180,E1 -11868.357,E2 -11868.357} C_VEL
LIN {X 0,Y 383.248,Z 733.931,A -85,B 0,C 180,E1 -11870.501,E2 -11870.501} C_VEL
LIN {X 0,Y 383.66,Z 731.414,A -85,B 0,C 180,E1 -11872.633,E2 -11872.633} C_VEL
LIN {X 0,Y 384.245,Z 727.416,A -85,B 0,C 180,E1 -11874.753,E2 -11874.753} C_VEL
LIN {X 0,Y 384.724,Z 723.352,A -85,B 0,C 180,E1 -11876.335,E2 -11876.335} C_VEL
LIN {X 0,Y 385.434,Z 718.268,A -85,B 0,C 180,E1 -11877.911,E2 -11877.911} C_VEL
LIN {X 0,Y 386.301,Z 710.95,A -85,B 0,C 180,E1 -11879.74,E2 -11879.74} C_VEL
LIN {X 0,Y 387.373,Z 702.086,A -85,B 0,C 180,E1 -11881.5,E2 -11881.5} C_VEL
LIN {X 0,Y 388.293,Z 693.756,A -85,B 0,C 180,E1 -11882.853,E2 -11882.853} C_VEL
LIN {X 0,Y 389.267,Z 683.185,A -85,B 0,C 180,E1 -11884.271,E2 -11884.271} C_VEL
LIN {X 0,Y 390.35,Z 671.373,A -85,B 0,C 180,E1 -11885.554,E2 -11885.554} C_VEL
LIN {X 0,Y 391.238,Z 659.639,A -85,B 0,C 180,E1 -11886.576,E2 -11886.576} C_VEL
LIN {X 0,Y 391.838,Z 646.686,A -85,B 0,C 180,E1 -11887.472,E2 -11887.472} C_VEL
LIN {X 0,Y 392.288,Z 633.692,A -85,B 0,C 180,E1 -11888.143,E2 -11888.143} C_VEL
LIN {X 0,Y 392.444,Z 619.803,A -85,B 0,C 180,E1 -11888.652,E2 -11888.652} C_VEL
LIN {X 0,Y 392.776,Z 587.984,A -85,B 0,C 180,E1 -11889.365,E2 -11889.365} C_VEL
LIN {X 0,Y 392.997,Z 573.912,A -85,B 0,C 180,E1 -11889.671,E2 -11889.671} C_VEL
LIN {X 0,Y 386.885,Z 560.763,A -85,B 0,C 180,E1 -11890.48,E2 -11890.48} C_VEL
LIN {X 0,Y 383.308,Z 553.615,A -85,B 0,C 180,E1 -11890.962,E2 -11890.962} C_VEL
LIN {X 0,Y 383.134,Z 552.762,A -85,B 0,C 180,E1 -11891.025,E2 -11891.025} C_VEL
LIN {X 0,Y 383.124,Z 552.767,A -85,B 0,C 180,E1 -11893.797,E2 -11893.797} C_VEL
LIN {X 0,Y 383.091,Z 552.77,A -85,B 0,C 180,E1 -11897.455,E2 -11897.455} C_VEL
LIN {X 0,Y 383.026,Z 552.774,A -85,B 0,C 180,E1 -11900.648,E2 -11900.648} C_VEL
LIN {X 0,Y 383.03,Z 552.773,A -85,B 0,C 180,E1 -11903.808,E2 -11903.808} C_VEL
LIN {X 0,Y 383.054,Z 552.767,A -85,B 0,C 180,E1 -11907.303,E2 -11907.303} C_VEL
LIN {X 0,Y 382.984,Z 552.773,A -85,B 0,C 180,E1 -11910.919,E2 -11910.919} C_VEL
LIN {X 0,Y 383.016,Z 552.766,A -85,B 0,C 180,E1 -11914.669,E2 -11914.669} C_VEL
LIN {X 0,Y 383,Z 552.774,A -85,B 0,C 180,E1 -11917.905,E2 -11917.905} C_VEL
LIN {X 0,Y 382.984,Z 552.777,A -85,B 0,C 180,E1 -11921.348,E2 -11921.348} C_VEL
LIN {X 0,Y 382.997,Z 552.774,A -85,B 0,C 180,E1 -11924.305,E2 -11924.305} C_VEL
LIN {X 0,Y 383.009,Z 552.778,A -85,B 0,C 180,E1 -11927.241,E2 -11927.241} C_VEL
LIN {X 0,Y 383.015,Z 552.774,A -85,B 0,C 180,E1 -11930.414,E2 -11930.414} C_VEL
LIN {X 0,Y 383.074,Z 552.865,A -85,B 0,C 180,E1 -11932.238,E2 -11932.238} C_VEL
LIN {X 0,Y 386.216,Z 567.851,A -85,B 0,C 180,E1 -11935.934,E2 -11935.934} C_VEL
LIN {X 0,Y 387.773,Z 575.168,A -85,B 0,C 180,E1 -11937.68,E2 -11937.68} C_VEL
LIN {X 0,Y 387.019,Z 584.548,A -85,B 0,C 180,E1 -11939.741,E2 -11939.741} C_VEL
LIN {X 0,Y 385.605,Z 600.792,A -85,B 0,C 180,E1 -11943.262,E2 -11943.262} C_VEL
LIN {X 0,Y 384.419,Z 617.593,A -85,B 0,C 180,E1 -11946.855,E2 -11946.855} C_VEL
LIN {X 0,Y 384.097,Z 623.948,A -85,B 0,C 180,E1 -11948.154,E2 -11948.154} C_VEL
LIN {X 0,Y 386.461,Z 643.115,A -85,B 0,C 180,E1 -11948.867,E2 -11948.867} C_VEL
LIN {X 0,Y 390.24,Z 676.662,A -85,B 0,C 180,E1 -11950.016,E2 -11950.016} C_VEL
LIN {X 0,Y 388.738,Z 733.883,A -85,B 0,C 180,E1 -11951.386,E2 -11951.386} C_VEL
LIN {X 0,Y 387.954,Z 748.117,A -85,B 0,C 180,E1 -11951.928,E2 -11951.928} C_VEL
LIN {X 0,Y 386.947,Z 762.142,A -85,B 0,C 180,E1 -11952.698,E2 -11952.698} C_VEL
LIN {X 0,Y 385.648,Z 776.784,A -85,B 0,C 180,E1 -11953.729,E2 -11953.729} C_VEL
LIN {X 0,Y 384.711,Z 788.482,A -85,B 0,C 180,E1 -11954.776,E2 -11954.776} C_VEL
LIN {X 0,Y 383.948,Z 799.187,A -85,B 0,C 180,E1 -11955.965,E2 -11955.965} C_VEL
LIN {X 0,Y 383.274,Z 808.976,A -85,B 0,C 180,E1 -11957.289,E2 -11957.289} C_VEL
LIN {X 0,Y 382.764,Z 817.082,A -85,B 0,C 180,E1 -11958.617,E2 -11958.617} C_VEL
LIN {X 0,Y 382.392,Z 825.07,A -85,B 0,C 180,E1 -11960.212,E2 -11960.212} C_VEL
LIN {X 0,Y 382.271,Z 830.542,A -85,B 0,C 180,E1 -11961.543,E2 -11961.543} C_VEL
LIN {X 0,Y 382.233,Z 835.905,A -85,B 0,C 180,E1 -11963.163,E2 -11963.163} C_VEL
LIN {X 0,Y 382.368,Z 839.907,A -85,B 0,C 180,E1 -11964.728,E2 -11964.728} C_VEL
LIN {X 0,Y 382.471,Z 841.966,A -85,B 0,C 180,E1 -11965.786,E2 -11965.786} C_VEL
LIN {X 0,Y 382.449,Z 843.541,A -85,B 0,C 180,E1 -11966.84,E2 -11966.84} C_VEL
LIN {X 0,Y 382.471,Z 844.67,A -85,B 0,C 180,E1 -11967.895,E2 -11967.895} C_VEL
LIN {X 0,Y 382.508,Z 845.329,A -85,B 0,C 180,E1 -11968.948,E2 -11968.948} C_VEL
LIN {X 0,Y 382.75,Z 845.543,A -85,B 0,C 180,E1 -11970.001,E2 -11970.001} C_VEL
LIN {X 0,Y 382.515,Z 845.243,A -85,B 0,C 180,E1 -11971.053,E2 -11971.053} C_VEL
LIN {X 0,Y 382.477,Z 844.533,A -85,B 0,C 180,E1 -11972.107,E2 -11972.107} C_VEL
LIN {X 0,Y 382.459,Z 843.368,A -85,B 0,C 180,E1 -11973.161,E2 -11973.161} C_VEL
LIN {X 0,Y 382.415,Z 840.74,A -85,B 0,C 180,E1 -11974.744,E2 -11974.744} C_VEL
LIN {X 0,Y 382.284,Z 837.006,A -85,B 0,C 180,E1 -11976.334,E2 -11976.334} C_VEL
LIN {X 0,Y 382.222,Z 832.118,A -85,B 0,C 180,E1 -11977.927,E2 -11977.927} C_VEL
LIN {X 0,Y 382.344,Z 824.812,A -85,B 0,C 180,E1 -11979.79,E2 -11979.79} C_VEL
LIN {X 0,Y 382.711,Z 816.981,A -85,B 0,C 180,E1 -11981.386,E2 -11981.386} C_VEL
LIN {X 0,Y 383.276,Z 807.665,A -85,B 0,C 180,E1 -11982.949,E2 -11982.949} C_VEL
LIN {X 0,Y 383.827,Z 800.097,A -85,B 0,C 180,E1 -11984.014,E2 -11984.014} C_VEL
LIN {X 0,Y 384.76,Z 788.803,A -85,B 0,C 180,E1 -11985.359,E2 -11985.359} C_VEL
LIN {X 0,Y 386.033,Z 776.649,A -85,B 0,C 180,E1 -11986.527,E2 -11986.527} C_VEL
LIN {X 0,Y 387.284,Z 763.236,A -85,B 0,C 180,E1 -11987.56,E2 -11987.56} C_VEL
LIN {X 0,Y 388.639,Z 749.447,A -85,B 0,C 180,E1 -11988.381,E2 -11988.381} C_VEL
LIN {X 0,Y 389.712,Z 734.351,A -85,B 0,C 180,E1 -11989.045,E2 -11989.045} C_VEL
LIN {X 0,Y 390.408,Z 718.565,A -85,B 0,C 180,E1 -11989.522,E2 -11989.522} C_VEL
LIN {X 0,Y 391.697,Z 676.015,A -85,B 0,C 180,E1 -11990.583,E2 -11990.583} C_VEL
LIN {X 0,Y 390.722,Z 657.995,A -85,B 0,C 180,E1 -11991.169,E2 -11991.169} C_VEL
LIN {X 0,Y 389.492,Z 639.072,A -85,B 0,C 180,E1 -11991.823,E2 -11991.823} C_VEL
LIN {X 0,Y 387.355,Z 620.636,A -85,B 0,C 180,E1 -11992.567,E2 -11992.567} C_VEL
LIN {X 0,Y 384.162,Z 602.21,A -85,B 0,C 180,E1 -11993.455,E2 -11993.455} C_VEL
LIN {X 0,Y 383.465,Z 597.537,A -85,B 0,C 180,E1 -11993.703,E2 -11993.703} C_VEL
LIN {X 0,Y 384.015,Z 580.121,A -85,B 0,C 180,E1 -11997.229,E2 -11997.229} C_VEL
LIN {X 0,Y 384.722,Z 564.699,A -85,B 0,C 180,E1 -12000.46,E2 -12000.46} C_VEL
LIN {X 0,Y 384.529,Z 560.492,A -85,B 0,C 180,E1 -12001.392,E2 -12001.392} C_VEL
LIN {X 0,Y 383.088,Z 552.771,A -85,B 0,C 180,E1 -12003.221,E2 -12003.221} C_VEL
LIN {X 0,Y 383.037,Z 552.771,A -85,B 0,C 180,E1 -12006.165,E2 -12006.165} C_VEL
LIN {X 0,Y 383.013,Z 552.773,A -85,B 0,C 180,E1 -12009.958,E2 -12009.958} C_VEL
LIN {X 0,Y 383.01,Z 552.776,A -85,B 0,C 180,E1 -12012.779,E2 -12012.779} C_VEL
LIN {X 0,Y 383.002,Z 552.776,A -85,B 0,C 180,E1 -12015.789,E2 -12015.789} C_VEL
LIN {X 0,Y 382.993,Z 552.777,A -85,B 0,C 180,E1 -12018.796,E2 -12018.796} C_VEL
LIN {X 0,Y 383.004,Z 552.776,A -85,B 0,C 180,E1 -12022.096,E2 -12022.096} C_VEL
LIN {X 0,Y 383.022,Z 552.775,A -85,B 0,C 180,E1 -12025.332,E2 -12025.332} C_VEL
LIN {X 0,Y 382.988,Z 552.779,A -85,B 0,C 180,E1 -12029.081,E2 -12029.081} C_VEL
LIN {X 0,Y 383.061,Z 552.772,A -85,B 0,C 180,E1 -12032.698,E2 -12032.698} C_VEL
LIN {X 0,Y 383.035,Z 552.777,A -85,B 0,C 180,E1 -12036.121,E2 -12036.121} C_VEL
LIN {X 0,Y 384.107,Z 555.726,A -85,B 0,C 180,E1 -12036.334,E2 -12036.334} C_VEL
LIN {X 0,Y 385.49,Z 557.957,A -85,B 0,C 180,E1 -12036.535,E2 -12036.535} C_VEL
LIN {X 0,Y 392.098,Z 570.364,A -85,B 0,C 180,E1 -12037.461,E2 -12037.461} C_VEL
LIN {X 0,Y 394.83,Z 576.468,A -85,B 0,C 180,E1 -12037.845,E2 -12037.845} C_VEL
LIN {X 0,Y 394.746,Z 608.95,A -85,B 0,C 180,E1 -12038.588,E2 -12038.588} C_VEL
LIN {X 0,Y 394.664,Z 623.704,A -85,B 0,C 180,E1 -12039.136,E2 -12039.136} C_VEL
LIN {X 0,Y 394.247,Z 637.753,A -85,B 0,C 180,E1 -12039.862,E2 -12039.862} C_VEL
LIN {X 0,Y 393.579,Z 650.5,A -85,B 0,C 180,E1 -12040.71,E2 -12040.71} C_VEL
LIN {X 0,Y 392.722,Z 663.068,A -85,B 0,C 180,E1 -12041.753,E2 -12041.753} C_VEL
LIN {X 0,Y 391.735,Z 674.517,A -85,B 0,C 180,E1 -12042.915,E2 -12042.915} C_VEL
LIN {X 0,Y 390.758,Z 684.122,A -85,B 0,C 180,E1 -12044.08,E2 -12044.08} C_VEL
LIN {X 0,Y 389.501,Z 694.818,A -85,B 0,C 180,E1 -12045.634,E2 -12045.634} C_VEL
LIN {X 0,Y 388.37,Z 703.732,A -85,B 0,C 180,E1 -12047.192,E2 -12047.192} C_VEL
LIN {X 0,Y 387.305,Z 711.626,A -85,B 0,C 180,E1 -12048.854,E2 -12048.854} C_VEL
LIN {X 0,Y 386.32,Z 718.381,A -85,B 0,C 180,E1 -12050.576,E2 -12050.576} C_VEL
LIN {X 0,Y 385.21,Z 724.986,A -85,B 0,C 180,E1 -12052.662,E2 -12052.662} C_VEL
LIN {X 0,Y 384.582,Z 729.973,A -85,B 0,C 180,E1 -12054.757,E2 -12054.757} C_VEL
LIN {X 0,Y 383.958,Z 733.614,A -85,B 0,C 180,E1 -12056.852,E2 -12056.852} C_VEL
LIN {X 0,Y 383.567,Z 735.94,A -85,B 0,C 180,E1 -12058.95,E2 -12058.95} C_VEL
LIN {X 0,Y 383.298,Z 737.031,A -85,B 0,C 180,E1 -12061.05,E2 -12061.05} C_VEL
LIN {X 0,Y 383.165,Z 736.901,A -85,B 0,C 180,E1 -12063.154,E2 -12063.154} C_VEL
LIN {X 0,Y 383.091,Z 735.561,A -85,B 0,C 180,E1 -12065.263,E2 -12065.263} C_VEL
LIN {X 0,Y 383.293,Z 733.986,A -85,B 0,C 180,E1 -12066.621,E2 -12066.621} C_VEL
LIN {X 0,Y 383.419,Z 730.215,A -85,B 0,C 180,E1 -12068.963,E2 -12068.963} C_VEL
LIN {X 0,Y 383.72,Z 725.294,A -85,B 0,C 180,E1 -12071.087,E2 -12071.087} C_VEL
LIN {X 0,Y 384.199,Z 718.847,A -85,B 0,C 180,E1 -12073.218,E2 -12073.218} C_VEL
LIN {X 0,Y 384.793,Z 711.81,A -85,B 0,C 180,E1 -12075.085,E2 -12075.085} C_VEL
LIN {X 0,Y 385.566,Z 703.211,A -85,B 0,C 180,E1 -12076.956,E2 -12076.956} C_VEL
LIN {X 0,Y 386.386,Z 693.906,A -85,B 0,C 180,E1 -12078.641,E2 -12078.641} C_VEL
LIN {X 0,Y 387.27,Z 682.863,A -85,B 0,C 180,E1 -12080.308,E2 -12080.308} C_VEL
LIN {X 0,Y 388.177,Z 671.073,A -85,B 0,C 180,E1 -12081.786,E2 -12081.786} C_VEL
LIN {X 0,Y 389.086,Z 659.092,A -85,B 0,C 180,E1 -12083.037,E2 -12083.037} C_VEL
LIN {X 0,Y 389.973,Z 645.473,A -85,B 0,C 180,E1 -12084.204,E2 -12084.204} C_VEL
LIN {X 0,Y 390.658,Z 631.751,A -85,B 0,C 180,E1 -12085.151,E2 -12085.151} C_VEL
LIN {X 0,Y 391.286,Z 616.374,A -85,B 0,C 180,E1 -12085.968,E2 -12085.968} C_VEL
LIN {X 0,Y 391.575,Z 600.675,A -85,B 0,C 180,E1 -12086.574,E2 -12086.574} C_VEL
LIN {X 0,Y 391.664,Z 575.929,A -85,B 0,C 180,E1 -12087.184,E2 -12087.184} C_VEL
LIN {X 0,Y 383.043,Z 552.773,A -85,B 0,C 180,E1 -12088.147,E2 -12088.147} C_VEL
LIN {X 0,Y 382.984,Z 552.775,A -85,B 0,C 180,E1 -12090.918,E2 -12090.918} C_VEL
LIN {X 0,Y 383.019,Z 552.772,A -85,B 0,C 180,E1 -12094.667,E2 -12094.667} C_VEL
LIN {X 0,Y 383,Z 552.776,A -85,B 0,C 180,E1 -12097.903,E2 -12097.903} C_VEL
LIN {X 0,Y 382.984,Z 552.775,A -85,B 0,C 180,E1 -12101.347,E2 -12101.347} C_VEL
LIN {X 0,Y 382.996,Z 552.781,A -85,B 0,C 180,E1 -12104.303,E2 -12104.303} C_VEL
LIN {X 0,Y 383.01,Z 552.771,A -85,B 0,C 180,E1 -12107.239,E2 -12107.239} C_VEL
LIN {X 0,Y 383.016,Z 552.778,A -85,B 0,C 180,E1 -12110.413,E2 -12110.413} C_VEL
LIN {X 0,Y 383.026,Z 552.772,A -85,B 0,C 180,E1 -12114.044,E2 -12114.044} C_VEL
LIN {X 0,Y 382.986,Z 552.774,A -85,B 0,C 180,E1 -12117.577,E2 -12117.577} C_VEL
LIN {X 0,Y 382.991,Z 552.777,A -85,B 0,C 180,E1 -12120.299,E2 -12120.299} C_VEL
LIN {X 0,Y 383.079,Z 552.764,A -85,B 0,C 180,E1 -12124.02,E2 -12124.02} C_VEL
LIN {X 0,Y 383.007,Z 552.773,A -85,B 0,C 180,E1 -12127.335,E2 -12127.335} C_VEL
LIN {X 0,Y 383.059,Z 552.772,A -85,B 0,C 180,E1 -12130.716,E2 -12130.716} C_VEL
LIN {X 0,Y 383.079,Z 552.763,A -85,B 0,C 180,E1 -12134.026,E2 -12134.026} C_VEL
LIN {X 0,Y 383.135,Z 552.759,A -85,B 0,C 180,E1 -12137.283,E2 -12137.283} C_VEL
LIN {X 0,Y 383.15,Z 552.756,A -85,B 0,C 180,E1 -12140.497,E2 -12140.497} C_VEL
LIN {X 0,Y 383.271,Z 552.742,A -85,B 0,C 180,E1 -12142.625,E2 -12142.625} C_VEL
LIN {X 0,Y 383.198,Z 552.752,A -85,B 0,C 180,E1 -12144.738,E2 -12144.738} C_VEL
LIN {X 0,Y 383.386,Z 552.725,A -85,B 0,C 180,E1 -12147.898,E2 -12147.898} C_VEL
LIN {X 0,Y 383.517,Z 552.708,A -85,B 0,C 180,E1 -12149.999,E2 -12149.999} C_VEL
LIN {X 0,Y 383.25,Z 552.748,A -85,B 0,C 180,E1 -12153.153,E2 -12153.153} C_VEL
LIN {X 0,Y 383.281,Z 552.738,A -85,B 0,C 180,E1 -12156.316,E2 -12156.316} C_VEL
LIN {X 0,Y 383.257,Z 552.741,A -85,B 0,C 180,E1 -12158.435,E2 -12158.435} C_VEL
LIN {X 0,Y 383.106,Z 552.763,A -85,B 0,C 180,E1 -12161.641,E2 -12161.641} C_VEL
LIN {X 0,Y 383.109,Z 552.761,A -85,B 0,C 180,E1 -12164.881,E2 -12164.881} C_VEL
LIN {X 0,Y 383.059,Z 552.766,A -85,B 0,C 180,E1 -12168.173,E2 -12168.173} C_VEL
LIN {X 0,Y 382.995,Z 552.781,A -85,B 0,C 180,E1 -12171.53,E2 -12171.53} C_VEL
LIN {X 0,Y 383.048,Z 552.768,A -85,B 0,C 180,E1 -12174.96,E2 -12174.96} C_VEL
LIN {X 0,Y 383.072,Z 552.766,A -85,B 0,C 180,E1 -12175.939,E2 -12175.939} C_VEL
LIN {X 0,Y 382.453,Z 552.849,A -85,B 0,C 180,E1 -12176.817,E2 -12176.817} C_VEL
LIN {X 0,Y 379.581,Z 553.207,A -85,B 0,C 180,E1 -12178.243,E2 -12178.243} C_VEL
LIN {X 0,Y 377.113,Z 553.51,A -85,B 0,C 180,E1 -12179.396,E2 -12179.396} C_VEL
LIN {X 0,Y 376.05,Z 553.64,A -85,B 0,C 180,E1 -12180.288,E2 -12180.288} C_VEL
LIN {X 0,Y 375.964,Z 553.649,A -85,B 0,C 180,E1 -12180.591,E2 -12180.591} C_VEL
LIN {X 0,Y 375.958,Z 553.653,A -85,B 0,C 180,E1 -12184.111,E2 -12184.111} C_VEL
LIN {X 0,Y 375.95,Z 553.651,A -85,B 0,C 180,E1 -12186.741,E2 -12186.741} C_VEL
LIN {X 0,Y 375.992,Z 553.652,A -85,B 0,C 180,E1 -12189.972,E2 -12189.972} C_VEL
LIN {X 0,Y 375.941,Z 553.657,A -85,B 0,C 180,E1 -12193.763,E2 -12193.763} C_VEL
LIN {X 0,Y 375.984,Z 553.647,A -85,B 0,C 180,E1 -12196.801,E2 -12196.801} C_VEL
LIN {X 0,Y 375.995,Z 553.652,A -85,B 0,C 180,E1 -12200.027,E2 -12200.027} C_VEL
LIN {X 0,Y 375.96,Z 553.651,A -85,B 0,C 180,E1 -12203.495,E2 -12203.495} C_VEL
LIN {X 0,Y 376.003,Z 553.651,A -85,B 0,C 180,E1 -12204.165,E2 -12204.165} C_VEL
LIN {X 0,Y 379.809,Z 564.201,A -85,B 0,C 180,E1 -12204.611,E2 -12204.611} C_VEL
LIN {X 0,Y 383.77,Z 574.791,A -85,B 0,C 180,E1 -12205.035,E2 -12205.035} C_VEL
LIN {X 0,Y 383.227,Z 614.56,A -85,B 0,C 180,E1 -12205.933,E2 -12205.933} C_VEL
LIN {X 0,Y 383.002,Z 628.714,A -85,B 0,C 180,E1 -12206.455,E2 -12206.455} C_VEL
LIN {X 0,Y 382.517,Z 642.599,A -85,B 0,C 180,E1 -12207.18,E2 -12207.18} C_VEL
LIN {X 0,Y 381.873,Z 655.275,A -85,B 0,C 180,E1 -12208.055,E2 -12208.055} C_VEL
LIN {X 0,Y 381.076,Z 668.539,A -85,B 0,C 180,E1 -12209.218,E2 -12209.218} C_VEL
LIN {X 0,Y 380.157,Z 680.807,A -85,B 0,C 180,E1 -12210.553,E2 -12210.553} C_VEL
LIN {X 0,Y 379.408,Z 690.306,A -85,B 0,C 180,E1 -12211.814,E2 -12211.814} C_VEL
LIN {X 0,Y 378.716,Z 699.323,A -85,B 0,C 180,E1 -12213.239,E2 -12213.239} C_VEL
LIN {X 0,Y 377.916,Z 708.407,A -85,B 0,C 180,E1 -12214.972,E2 -12214.972} C_VEL
LIN {X 0,Y 377.29,Z 715.729,A -85,B 0,C 180,E1 -12216.682,E2 -12216.682} C_VEL
LIN {X 0,Y 376.706,Z 722.416,A -85,B 0,C 180,E1 -12218.621,E2 -12218.621} C_VEL
LIN {X 0,Y 376.373,Z 727.146,A -85,B 0,C 180,E1 -12220.36,E2 -12220.36} C_VEL
LIN {X 0,Y 376.078,Z 731.293,A -85,B 0,C 180,E1 -12222.374,E2 -12222.374} C_VEL
LIN {X 0,Y 375.931,Z 733.348,A -85,B 0,C 180,E1 -12223.715,E2 -12223.715} C_VEL
LIN {X 0,Y 375.887,Z 735.439,A -85,B 0,C 180,E1 -12225.933,E2 -12225.933} C_VEL
LIN {X 0,Y 376.017,Z 736.065,A -85,B 0,C 180,E1 -12228.136,E2 -12228.136} C_VEL
LIN {X 0,Y 376.241,Z 735.267,A -85,B 0,C 180,E1 -12230.322,E2 -12230.322} C_VEL
LIN {X 0,Y 376.65,Z 732.978,A -85,B 0,C 180,E1 -12232.495,E2 -12232.495} C_VEL
LIN {X 0,Y 377.255,Z 729.183,A -85,B 0,C 180,E1 -12234.656,E2 -12234.656} C_VEL
LIN {X 0,Y 377.99,Z 723.829,A -85,B 0,C 180,E1 -12236.803,E2 -12236.803} C_VEL
LIN {X 0,Y 378.879,Z 717.608,A -85,B 0,C 180,E1 -12238.672,E2 -12238.672} C_VEL
LIN {X 0,Y 379.783,Z 709.958,A -85,B 0,C 180,E1 -12240.496,E2 -12240.496} C_VEL
LIN {X 0,Y 380.929,Z 701.526,A -85,B 0,C 180,E1 -12242.115,E2 -12242.115} C_VEL
LIN {X 0,Y 382.023,Z 691.547,A -85,B 0,C 180,E1 -12243.692,E2 -12243.692} C_VEL
LIN {X 0,Y 383.101,Z 681.353,A -85,B 0,C 180,E1 -12245,E2 -12245} C_VEL
LIN {X 0,Y 384.038,Z 670.175,A -85,B 0,C 180,E1 -12246.172,E2 -12246.172} C_VEL
LIN {X 0,Y 384.958,Z 657.735,A -85,B 0,C 180,E1 -12247.211,E2 -12247.211} C_VEL
LIN {X 0,Y 385.545,Z 644.895,A -85,B 0,C 180,E1 -12248.056,E2 -12248.056} C_VEL
LIN {X 0,Y 385.984,Z 631.057,A -85,B 0,C 180,E1 -12248.735,E2 -12248.735} C_VEL
LIN {X 0,Y 386.067,Z 617.679,A -85,B 0,C 180,E1 -12249.183,E2 -12249.183} C_VEL
LIN {X 0,Y 386.723,Z 575.859,A -85,B 0,C 180,E1 -12250.121,E2 -12250.121} C_VEL
LIN {X 0,Y 380.31,Z 562.433,A -85,B 0,C 180,E1 -12251,E2 -12251} C_VEL
LIN {X 0,Y 377.046,Z 556.449,A -85,B 0,C 180,E1 -12251.455,E2 -12251.455} C_VEL
LIN {X 0,Y 376.059,Z 553.645,A -85,B 0,C 180,E1 -12251.638,E2 -12251.638} C_VEL
LIN {X 0,Y 376.063,Z 553.647,A -85,B 0,C 180,E1 -12254.061,E2 -12254.061} C_VEL
LIN {X 0,Y 376.041,Z 553.647,A -85,B 0,C 180,E1 -12257.608,E2 -12257.608} C_VEL
LIN {X 0,Y 375.975,Z 553.653,A -85,B 0,C 180,E1 -12260.833,E2 -12260.833} C_VEL
LIN {X 0,Y 375.991,Z 553.649,A -85,B 0,C 180,E1 -12264.282,E2 -12264.282} C_VEL
LIN {X 0,Y 376.017,Z 553.644,A -85,B 0,C 180,E1 -12266.653,E2 -12266.653} C_VEL
LIN {X 0,Y 375.974,Z 553.649,A -85,B 0,C 180,E1 -12269.079,E2 -12269.079} C_VEL
LIN {X 0,Y 375.947,Z 553.646,A -85,B 0,C 180,E1 -12272.829,E2 -12272.829} C_VEL
LIN {X 0,Y 375.956,Z 553.649,A -85,B 0,C 180,E1 -12275.416,E2 -12275.416} C_VEL
LIN {X 0,Y 375.974,Z 553.648,A -85,B 0,C 180,E1 -12278.272,E2 -12278.272} C_VEL
LIN {X 0,Y 375.934,Z 553.653,A -85,B 0,C 180,E1 -12281.602,E2 -12281.602} C_VEL
LIN {X 0,Y 375.952,Z 553.657,A -85,B 0,C 180,E1 -12285.265,E2 -12285.265} C_VEL
LIN {X 0,Y 375.939,Z 553.649,A -85,B 0,C 180,E1 -12289.134,E2 -12289.134} C_VEL
LIN {X 0,Y 376.018,Z 553.792,A -85,B 0,C 180,E1 -12292.004,E2 -12292.004} C_VEL
LIN {X 0,Y 379.282,Z 569.327,A -85,B 0,C 180,E1 -12295.909,E2 -12295.909} C_VEL
LIN {X 0,Y 380.794,Z 576.478,A -85,B 0,C 180,E1 -12297.641,E2 -12297.641} C_VEL
LIN {X 0,Y 379.686,Z 589.048,A -85,B 0,C 180,E1 -12300.456,E2 -12300.456} C_VEL
LIN {X 0,Y 378.159,Z 606.97,A -85,B 0,C 180,E1 -12304.4,E2 -12304.4} C_VEL
LIN {X 0,Y 377.158,Z 621.201,A -85,B 0,C 180,E1 -12307.502,E2 -12307.502} C_VEL
LIN {X 0,Y 379.292,Z 636.329,A -85,B 0,C 180,E1 -12308.122,E2 -12308.122} C_VEL
LIN {X 0,Y 383.781,Z 677.374,A -85,B 0,C 180,E1 -12309.596,E2 -12309.596} C_VEL
LIN {X 0,Y 382.189,Z 732.492,A -85,B 0,C 180,E1 -12310.95,E2 -12310.95} C_VEL
LIN {X 0,Y 381.329,Z 747.325,A -85,B 0,C 180,E1 -12311.533,E2 -12311.533} C_VEL
LIN {X 0,Y 380.294,Z 761.101,A -85,B 0,C 180,E1 -12312.316,E2 -12312.316} C_VEL
LIN {X 0,Y 379.177,Z 772.753,A -85,B 0,C 180,E1 -12313.166,E2 -12313.166} C_VEL
LIN {X 0,Y 378.014,Z 784.258,A -85,B 0,C 180,E1 -12314.223,E2 -12314.223} C_VEL
LIN {X 0,Y 376.987,Z 797.457,A -85,B 0,C 180,E1 -12315.7,E2 -12315.7} C_VEL
LIN {X 0,Y 376.319,Z 807.36,A -85,B 0,C 180,E1 -12317.05,E2 -12317.05} C_VEL
LIN {X 0,Y 375.745,Z 815.558,A -85,B 0,C 180,E1 -12318.401,E2 -12318.401} C_VEL
LIN {X 0,Y 375.323,Z 823.666,A -85,B 0,C 180,E1 -12320.026,E2 -12320.026} C_VEL
LIN {X 0,Y 375.22,Z 829.19,A -85,B 0,C 180,E1 -12321.383,E2 -12321.383} C_VEL
LIN {X 0,Y 375.177,Z 834.928,A -85,B 0,C 180,E1 -12323.134,E2 -12323.134} C_VEL
LIN {X 0,Y 375.326,Z 838.704,A -85,B 0,C 180,E1 -12324.628,E2 -12324.628} C_VEL
LIN {X 0,Y 375.441,Z 840.812,A -85,B 0,C 180,E1 -12325.706,E2 -12325.706} C_VEL
LIN {X 0,Y 375.42,Z 842.41,A -85,B 0,C 180,E1 -12326.781,E2 -12326.781} C_VEL
LIN {X 0,Y 375.444,Z 843.561,A -85,B 0,C 180,E1 -12327.855,E2 -12327.855} C_VEL
LIN {X 0,Y 375.509,Z 844.264,A -85,B 0,C 180,E1 -12328.928,E2 -12328.928} C_VEL
LIN {X 0,Y 375.725,Z 844.495,A -85,B 0,C 180,E1 -12330.001,E2 -12330.001} C_VEL
LIN {X 0,Y 375.485,Z 844.211,A -85,B 0,C 180,E1 -12331.073,E2 -12331.073} C_VEL
LIN {X 0,Y 375.439,Z 843.512,A -85,B 0,C 180,E1 -12332.146,E2 -12332.146} C_VEL
LIN {X 0,Y 375.414,Z 842.374,A -85,B 0,C 180,E1 -12333.22,E2 -12333.22} C_VEL
LIN {X 0,Y 375.345,Z 839.757,A -85,B 0,C 180,E1 -12334.834,E2 -12334.834} C_VEL
LIN {X 0,Y 375.208,Z 836.052,A -85,B 0,C 180,E1 -12336.453,E2 -12336.453} C_VEL
LIN {X 0,Y 375.145,Z 831.197,A -85,B 0,C 180,E1 -12338.078,E2 -12338.078} C_VEL
LIN {X 0,Y 375.268,Z 823.963,A -85,B 0,C 180,E1 -12339.976,E2 -12339.976} C_VEL
LIN {X 0,Y 375.688,Z 816.201,A -85,B 0,C 180,E1 -12341.602,E2 -12341.602} C_VEL
LIN {X 0,Y 376.236,Z 807.124,A -85,B 0,C 180,E1 -12343.168,E2 -12343.168} C_VEL
LIN {X 0,Y 376.948,Z 799.301,A -85,B 0,C 180,E1 -12344.303,E2 -12344.303} C_VEL
LIN {X 0,Y 377.893,Z 788.338,A -85,B 0,C 180,E1 -12345.645,E2 -12345.645} C_VEL
LIN {X 0,Y 379.206,Z 776.454,A -85,B 0,C 180,E1 -12346.834,E2 -12346.834} C_VEL
LIN {X 0,Y 380.533,Z 763.391,A -85,B 0,C 180,E1 -12347.882,E2 -12347.882} C_VEL
LIN {X 0,Y 382.031,Z 748.97,A -85,B 0,C 180,E1 -12348.781,E2 -12348.781} C_VEL
LIN {X 0,Y 383.195,Z 734.532,A -85,B 0,C 180,E1 -12349.451,E2 -12349.451} C_VEL
LIN {X 0,Y 383.981,Z 718.79,A -85,B 0,C 180,E1 -12349.967,E2 -12349.967} C_VEL
LIN {X 0,Y 385.382,Z 676.859,A -85,B 0,C 180,E1 -12351.046,E2 -12351.046} C_VEL
LIN {X 0,Y 383.573,Z 642.168,A -85,B 0,C 180,E1 -12352.239,E2 -12352.239} C_VEL
LIN {X 0,Y 381.191,Z 621.26,A -85,B 0,C 180,E1 -12353.123,E2 -12353.123} C_VEL
LIN {X 0,Y 378.25,Z 604.098,A -85,B 0,C 180,E1 -12353.981,E2 -12353.981} C_VEL
LIN {X 0,Y 376.511,Z 594.326,A -85,B 0,C 180,E1 -12354.51,E2 -12354.51} C_VEL
LIN {X 0,Y 377.191,Z 575.896,A -85,B 0,C 180,E1 -12358.368,E2 -12358.368} C_VEL
LIN {X 0,Y 377.767,Z 564.867,A -85,B 0,C 180,E1 -12360.756,E2 -12360.756} C_VEL
LIN {X 0,Y 377.357,Z 560.545,A -85,B 0,C 180,E1 -12361.745,E2 -12361.745} C_VEL
LIN {X 0,Y 376.06,Z 553.646,A -85,B 0,C 180,E1 -12363.457,E2 -12363.457} C_VEL
LIN {X 0,Y 375.958,Z 553.654,A -85,B 0,C 180,E1 -12366.741,E2 -12366.741} C_VEL
LIN {X 0,Y 375.993,Z 553.647,A -85,B 0,C 180,E1 -12369.971,E2 -12369.971} C_VEL
LIN {X 0,Y 375.934,Z 553.655,A -85,B 0,C 180,E1 -12373.766,E2 -12373.766} C_VEL
LIN {X 0,Y 375.938,Z 553.656,A -85,B 0,C 180,E1 -12376.811,E2 -12376.811} C_VEL
LIN {X 0,Y 375.967,Z 553.651,A -85,B 0,C 180,E1 -12380.537,E2 -12380.537} C_VEL
LIN {X 0,Y 375.968,Z 553.653,A -85,B 0,C 180,E1 -12383.495,E2 -12383.495} C_VEL
LIN {X 0,Y 375.964,Z 553.653,A -85,B 0,C 180,E1 -12385.888,E2 -12385.888} C_VEL
LIN {X 0,Y 375.969,Z 553.652,A -85,B 0,C 180,E1 -12389.687,E2 -12389.687} C_VEL
LIN {X 0,Y 376.024,Z 553.65,A -85,B 0,C 180,E1 -12393.348,E2 -12393.348} C_VEL
LIN {X 0,Y 376.03,Z 553.773,A -85,B 0,C 180,E1 -12395.4,E2 -12395.4} C_VEL
LIN {X 0,Y 377.146,Z 556.73,A -85,B 0,C 180,E1 -12395.61,E2 -12395.61} C_VEL
LIN {X 0,Y 378.498,Z 558.778,A -85,B 0,C 180,E1 -12395.814,E2 -12395.814} C_VEL
LIN {X 0,Y 384.186,Z 569.095,A -85,B 0,C 180,E1 -12396.682,E2 -12396.682} C_VEL
LIN {X 0,Y 388.852,Z 578.845,A -85,B 0,C 180,E1 -12397.36,E2 -12397.36} C_VEL
LIN {X 0,Y 388.562,Z 608.557,A -85,B 0,C 180,E1 -12398.056,E2 -12398.056} C_VEL
LIN {X 0,Y 388.542,Z 623.578,A -85,B 0,C 180,E1 -12398.593,E2 -12398.593} C_VEL
LIN {X 0,Y 388.114,Z 637.986,A -85,B 0,C 180,E1 -12399.322,E2 -12399.322} C_VEL
LIN {X 0,Y 387.351,Z 651.82,A -85,B 0,C 180,E1 -12400.249,E2 -12400.249} C_VEL
LIN {X 0,Y 386.461,Z 664.029,A -85,B 0,C 180,E1 -12401.28,E2 -12401.28} C_VEL
LIN {X 0,Y 385.238,Z 676.861,A -85,B 0,C 180,E1 -12402.618,E2 -12402.618} C_VEL
LIN {X 0,Y 384.248,Z 686.352,A -85,B 0,C 180,E1 -12403.803,E2 -12403.803} C_VEL
LIN {X 0,Y 382.904,Z 696.896,A -85,B 0,C 180,E1 -12405.382,E2 -12405.382} C_VEL
LIN {X 0,Y 381.701,Z 705.662,A -85,B 0,C 180,E1 -12406.964,E2 -12406.964} C_VEL
LIN {X 0,Y 380.57,Z 713.409,A -85,B 0,C 180,E1 -12408.654,E2 -12408.654} C_VEL
LIN {X 0,Y 379.531,Z 720.073,A -85,B 0,C 180,E1 -12410.406,E2 -12410.406} C_VEL
LIN {X 0,Y 378.366,Z 726.586,A -85,B 0,C 180,E1 -12412.529,E2 -12412.529} C_VEL
LIN {X 0,Y 377.868,Z 730.338,A -85,B 0,C 180,E1 -12414.128,E2 -12414.128} C_VEL
LIN {X 0,Y 377.38,Z 733.38,A -85,B 0,C 180,E1 -12415.727,E2 -12415.727} C_VEL
LIN {X 0,Y 376.806,Z 736.244,A -85,B 0,C 180,E1 -12417.862,E2 -12417.862} C_VEL
LIN {X 0,Y 376.421,Z 737.852,A -85,B 0,C 180,E1 -12420,E2 -12420} C_VEL
LIN {X 0,Y 376.222,Z 738.226,A -85,B 0,C 180,E1 -12422.141,E2 -12422.141} C_VEL
LIN {X 0,Y 375.991,Z 737.396,A -85,B 0,C 180,E1 -12424.287,E2 -12424.287} C_VEL
LIN {X 0,Y 376.294,Z 735.035,A -85,B 0,C 180,E1 -12426.61,E2 -12426.61} C_VEL
LIN {X 0,Y 376.339,Z 731.945,A -85,B 0,C 180,E1 -12428.592,E2 -12428.592} C_VEL
LIN {X 0,Y 376.65,Z 727.235,A -85,B 0,C 180,E1 -12430.753,E2 -12430.753} C_VEL
LIN {X 0,Y 377.052,Z 721.045,A -85,B 0,C 180,E1 -12432.924,E2 -12432.924} C_VEL
LIN {X 0,Y 377.605,Z 714.663,A -85,B 0,C 180,E1 -12434.711,E2 -12434.711} C_VEL
LIN {X 0,Y 378.419,Z 705.896,A -85,B 0,C 180,E1 -12436.73,E2 -12436.73} C_VEL
LIN {X 0,Y 379.324,Z 696.209,A -85,B 0,C 180,E1 -12438.562,E2 -12438.562} C_VEL
LIN {X 0,Y 380.229,Z 685.3,A -85,B 0,C 180,E1 -12440.277,E2 -12440.277} C_VEL
LIN {X 0,Y 381.174,Z 673.778,A -85,B 0,C 180,E1 -12441.78,E2 -12441.78} C_VEL
LIN {X 0,Y 382.119,Z 661.329,A -85,B 0,C 180,E1 -12443.13,E2 -12443.13} C_VEL
LIN {X 0,Y 382.98,Z 648.916,A -85,B 0,C 180,E1 -12444.242,E2 -12444.242} C_VEL
LIN {X 0,Y 383.73,Z 634.711,A -85,B 0,C 180,E1 -12445.275,E2 -12445.275} C_VEL
LIN {X 0,Y 384.404,Z 619.951,A -85,B 0,C 180,E1 -12446.104,E2 -12446.104} C_VEL
LIN {X 0,Y 384.745,Z 604.815,A -85,B 0,C 180,E1 -12446.737,E2 -12446.737} C_VEL
LIN {X 0,Y 384.875,Z 588.317,A -85,B 0,C 180,E1 -12447.198,E2 -12447.198} C_VEL
LIN {X 0,Y 384.9,Z 577.652,A -85,B 0,C 180,E1 -12447.448,E2 -12447.448} C_VEL
LIN {X 0,Y 375.987,Z 553.651,A -85,B 0,C 180,E1 -12448.472,E2 -12448.472} C_VEL
LIN {X 0,Y 375.959,Z 553.651,A -85,B 0,C 180,E1 -12451.561,E2 -12451.561} C_VEL
LIN {X 0,Y 375.958,Z 553.65,A -85,B 0,C 180,E1 -12455.415,E2 -12455.415} C_VEL
LIN {X 0,Y 375.974,Z 553.654,A -85,B 0,C 180,E1 -12458.27,E2 -12458.27} C_VEL
LIN {X 0,Y 375.934,Z 553.654,A -85,B 0,C 180,E1 -12461.6,E2 -12461.6} C_VEL
LIN {X 0,Y 375.927,Z 553.654,A -85,B 0,C 180,E1 -12465.268,E2 -12465.268} C_VEL
LIN {X 0,Y 375.935,Z 553.66,A -85,B 0,C 180,E1 -12468.398,E2 -12468.398} C_VEL
LIN {X 0,Y 375.976,Z 553.648,A -85,B 0,C 180,E1 -12471.728,E2 -12471.728} C_VEL
LIN {X 0,Y 375.979,Z 553.647,A -85,B 0,C 180,E1 -12475.332,E2 -12475.332} C_VEL
LIN {X 0,Y 375.957,Z 553.656,A -85,B 0,C 180,E1 -12478.437,E2 -12478.437} C_VEL
LIN {X 0,Y 375.982,Z 553.649,A -85,B 0,C 180,E1 -12482.14,E2 -12482.14} C_VEL
LIN {X 0,Y 376.006,Z 553.649,A -85,B 0,C 180,E1 -12484.538,E2 -12484.538} C_VEL
LIN {X 0,Y 375.962,Z 553.65,A -85,B 0,C 180,E1 -12488.045,E2 -12488.045} C_VEL
LIN {X 0,Y 376.008,Z 553.644,A -85,B 0,C 180,E1 -12491.473,E2 -12491.473} C_VEL
LIN {X 0,Y 376.057,Z 553.644,A -85,B 0,C 180,E1 -12494.832,E2 -12494.832} C_VEL
LIN {X 0,Y 376.048,Z 553.639,A -85,B 0,C 180,E1 -12498.136,E2 -12498.136} C_VEL
LIN {X 0,Y 376.256,Z 553.613,A -85,B 0,C 180,E1 -12501.876,E2 -12501.876} C_VEL
LIN {X 0,Y 376.17,Z 553.626,A -85,B 0,C 180,E1 -12504.639,E2 -12504.639} C_VEL
LIN {X 0,Y 376.352,Z 553.601,A -85,B 0,C 180,E1 -12507.859,E2 -12507.859} C_VEL
LIN {X 0,Y 376.487,Z 553.584,A -85,B 0,C 180,E1 -12509.999,E2 -12509.999} C_VEL
LIN {X 0,Y 376.188,Z 553.628,A -85,B 0,C 180,E1 -12513.212,E2 -12513.212} C_VEL
LIN {X 0,Y 376.241,Z 553.615,A -85,B 0,C 180,E1 -12516.434,E2 -12516.434} C_VEL
LIN {X 0,Y 376.203,Z 553.62,A -85,B 0,C 180,E1 -12518.594,E2 -12518.594} C_VEL
LIN {X 0,Y 376.057,Z 553.639,A -85,B 0,C 180,E1 -12521.862,E2 -12521.862} C_VEL
LIN {X 0,Y 376.057,Z 553.642,A -85,B 0,C 180,E1 -12525.167,E2 -12525.167} C_VEL
LIN {X 0,Y 376.005,Z 553.644,A -85,B 0,C 180,E1 -12528.526,E2 -12528.526} C_VEL
LIN {X 0,Y 375.964,Z 553.652,A -85,B 0,C 180,E1 -12531.953,E2 -12531.953} C_VEL
LIN {X 0,Y 376.002,Z 553.65,A -85,B 0,C 180,E1 -12535.461,E2 -12535.461} C_VEL
LIN {X 0,Y 375.977,Z 553.649,A -85,B 0,C 180,E1 -12539.078,E2 -12539.078} C_VEL
LIN {X 0,Y 375.964,Z 553.649,A -85,B 0,C 180,E1 -12540.591,E2 -12540.591} C_VEL
LIN {X 0,Y 375.302,Z 553.737,A -85,B 0,C 180,E1 -12541.485,E2 -12541.485} C_VEL
LIN {X 0,Y 372.461,Z 554.086,A -85,B 0,C 180,E1 -12542.939,E2 -12542.939} C_VEL
LIN {X 0,Y 370.046,Z 554.389,A -85,B 0,C 180,E1 -12544.114,E2 -12544.114} C_VEL
LIN {X 0,Y 368.997,Z 554.517,A -85,B 0,C 180,E1 -12545.023,E2 -12545.023} C_VEL
LIN {X 0,Y 368.905,Z 554.527,A -85,B 0,C 180,E1 -12545.331,E2 -12545.331} C_VEL
LIN {X 0,Y 368.902,Z 554.529,A -85,B 0,C 180,E1 -12548.952,E2 -12548.952} C_VEL
LIN {X 0,Y 368.904,Z 554.534,A -85,B 0,C 180,E1 -12552.014,E2 -12552.014} C_VEL
LIN {X 0,Y 368.95,Z 554.523,A -85,B 0,C 180,E1 -12555.187,E2 -12555.187} C_VEL
LIN {X 0,Y 368.941,Z 554.529,A -85,B 0,C 180,E1 -12558.186,E2 -12558.186} C_VEL
LIN {X 0,Y 368.908,Z 554.529,A -85,B 0,C 180,E1 -12561.359,E2 -12561.359} C_VEL
LIN {X 0,Y 368.942,Z 554.57,A -85,B 0,C 180,E1 -12563.845,E2 -12563.845} C_VEL
LIN {X 0,Y 377.009,Z 576.361,A -85,B 0,C 180,E1 -12564.752,E2 -12564.752} C_VEL
LIN {X 0,Y 376.428,Z 615.15,A -85,B 0,C 180,E1 -12565.643,E2 -12565.643} C_VEL
LIN {X 0,Y 376.196,Z 629.45,A -85,B 0,C 180,E1 -12566.176,E2 -12566.176} C_VEL
LIN {X 0,Y 375.687,Z 643.315,A -85,B 0,C 180,E1 -12566.907,E2 -12566.907} C_VEL
LIN {X 0,Y 375.034,Z 656.117,A -85,B 0,C 180,E1 -12567.802,E2 -12567.802} C_VEL
LIN {X 0,Y 374.246,Z 668.641,A -85,B 0,C 180,E1 -12568.908,E2 -12568.908} C_VEL
LIN {X 0,Y 373.341,Z 680.9,A -85,B 0,C 180,E1 -12570.248,E2 -12570.248} C_VEL
LIN {X 0,Y 372.462,Z 691.75,A -85,B 0,C 180,E1 -12571.701,E2 -12571.701} C_VEL
LIN {X 0,Y 371.628,Z 701.594,A -85,B 0,C 180,E1 -12573.312,E2 -12573.312} C_VEL
LIN {X 0,Y 370.863,Z 710.378,A -85,B 0,C 180,E1 -12575.062,E2 -12575.062} C_VEL
LIN {X 0,Y 370.129,Z 718.621,A -85,B 0,C 180,E1 -12577.093,E2 -12577.093} C_VEL
LIN {X 0,Y 369.652,Z 724.229,A -85,B 0,C 180,E1 -12578.824,E2 -12578.824} C_VEL
LIN {X 0,Y 369.308,Z 728.687,A -85,B 0,C 180,E1 -12580.548,E2 -12580.548} C_VEL
LIN {X 0,Y 369.07,Z 732.124,A -85,B 0,C 180,E1 -12582.262,E2 -12582.262} C_VEL
LIN {X 0,Y 368.855,Z 735.294,A -85,B 0,C 180,E1 -12584.53,E2 -12584.53} C_VEL
LIN {X 0,Y 368.903,Z 736.668,A -85,B 0,C 180,E1 -12586.31,E2 -12586.31} C_VEL
LIN {X 0,Y 368.979,Z 737.14,A -85,B 0,C 180,E1 -12587.906,E2 -12587.906} C_VEL
LIN {X 0,Y 369.214,Z 736.542,A -85,B 0,C 180,E1 -12590.136,E2 -12590.136} C_VEL
LIN {X 0,Y 369.639,Z 734.514,A -85,B 0,C 180,E1 -12592.352,E2 -12592.352} C_VEL
LIN {X 0,Y 369.893,Z 732.947,A -85,B 0,C 180,E1 -12593.455,E2 -12593.455} C_VEL
LIN {X 0,Y 370.616,Z 728.579,A -85,B 0,C 180,E1 -12595.65,E2 -12595.65} C_VEL
LIN {X 0,Y 371.523,Z 722.589,A -85,B 0,C 180,E1 -12597.832,E2 -12597.832} C_VEL
LIN {X 0,Y 372.483,Z 715.921,A -85,B 0,C 180,E1 -12599.702,E2 -12599.702} C_VEL
LIN {X 0,Y 373.498,Z 708.602,A -85,B 0,C 180,E1 -12601.348,E2 -12601.348} C_VEL
LIN {X 0,Y 374.718,Z 699.796,A -85,B 0,C 180,E1 -12602.957,E2 -12602.957} C_VEL
LIN {X 0,Y 375.638,Z 691.075,A -85,B 0,C 180,E1 -12604.292,E2 -12604.292} C_VEL
LIN {X 0,Y 376.787,Z 680.462,A -85,B 0,C 180,E1 -12605.62,E2 -12605.62} C_VEL
LIN {X 0,Y 377.829,Z 668.843,A -85,B 0,C 180,E1 -12606.811,E2 -12606.811} C_VEL
LIN {X 0,Y 378.753,Z 655.907,A -85,B 0,C 180,E1 -12607.866,E2 -12607.866} C_VEL
LIN {X 0,Y 379.346,Z 642.556,A -85,B 0,C 180,E1 -12608.699,E2 -12608.699} C_VEL
LIN {X 0,Y 379.711,Z 628.56,A -85,B 0,C 180,E1 -12609.333,E2 -12609.333} C_VEL
LIN {X 0,Y 379.804,Z 613.717,A -85,B 0,C 180,E1 -12609.769,E2 -12609.769} C_VEL
LIN {X 0,Y 380.488,Z 577.956,A -85,B 0,C 180,E1 -12610.583,E2 -12610.583} C_VEL
LIN {X 0,Y 373.864,Z 564.225,A -85,B 0,C 180,E1 -12611.543,E2 -12611.543} C_VEL
LIN {X 0,Y 370.232,Z 557.707,A -85,B 0,C 180,E1 -12612.078,E2 -12612.078} C_VEL
LIN {X 0,Y 369.085,Z 554.946,A -85,B 0,C 180,E1 -12612.274,E2 -12612.274} C_VEL
LIN {X 0,Y 369.033,Z 554.52,A -85,B 0,C 180,E1 -12612.302,E2 -12612.302} C_VEL
LIN {X 0,Y 368.995,Z 554.527,A -85,B 0,C 180,E1 -12615.465,E2 -12615.465} C_VEL
LIN {X 0,Y 368.979,Z 554.526,A -85,B 0,C 180,E1 -12618.893,E2 -12618.893} C_VEL
LIN {X 0,Y 368.929,Z 554.53,A -85,B 0,C 180,E1 -12622.396,E2 -12622.396} C_VEL
LIN {X 0,Y 368.997,Z 554.518,A -85,B 0,C 180,E1 -12625.981,E2 -12625.981} C_VEL
LIN {X 0,Y 368.965,Z 554.52,A -85,B 0,C 180,E1 -12628.814,E2 -12628.814} C_VEL
LIN {X 0,Y 368.897,Z 554.522,A -85,B 0,C 180,E1 -12632.239,E2 -12632.239} C_VEL
LIN {X 0,Y 368.927,Z 554.521,A -85,B 0,C 180,E1 -12635.002,E2 -12635.002} C_VEL
LIN {X 0,Y 368.909,Z 554.529,A -85,B 0,C 180,E1 -12638.642,E2 -12638.642} C_VEL
LIN {X 0,Y 368.88,Z 554.531,A -85,B 0,C 180,E1 -12642.01,E2 -12642.01} C_VEL
LIN {X 0,Y 368.925,Z 554.533,A -85,B 0,C 180,E1 -12645.184,E2 -12645.184} C_VEL
LIN {X 0,Y 368.882,Z 554.531,A -85,B 0,C 180,E1 -12648.178,E2 -12648.178} C_VEL
LIN {X 0,Y 368.99,Z 554.64,A -85,B 0,C 180,E1 -12651.757,E2 -12651.757} C_VEL
LIN {X 0,Y 372.31,Z 570.672,A -85,B 0,C 180,E1 -12655.863,E2 -12655.863} C_VEL
LIN {X 0,Y 373.812,Z 578.508,A -85,B 0,C 180,E1 -12657.784,E2 -12657.784} C_VEL
LIN {X 0,Y 372.137,Z 594.949,A -85,B 0,C 180,E1 -12661.52,E2 -12661.52} C_VEL
LIN {X 0,Y 370.716,Z 612.032,A -85,B 0,C 180,E1 -12665.351,E2 -12665.351} C_VEL
LIN {X 0,Y 370.265,Z 618.557,A -85,B 0,C 180,E1 -12666.806,E2 -12666.806} C_VEL
LIN {X 0,Y 371.651,Z 627.191,A -85,B 0,C 180,E1 -12667.206,E2 -12667.206} C_VEL
LIN {X 0,Y 373.251,Z 639.521,A -85,B 0,C 180,E1 -12667.713,E2 -12667.713} C_VEL
LIN {X 0,Y 377.351,Z 678.374,A -85,B 0,C 180,E1 -12669.152,E2 -12669.152} C_VEL
LIN {X 0,Y 375.702,Z 731.285,A -85,B 0,C 180,E1 -12670.502,E2 -12670.502} C_VEL
LIN {X 0,Y 374.846,Z 745.312,A -85,B 0,C 180,E1 -12671.06,E2 -12671.06} C_VEL
LIN {X 0,Y 373.681,Z 759.267,A -85,B 0,C 180,E1 -12671.851,E2 -12671.851} C_VEL
LIN {X 0,Y 372.366,Z 772.582,A -85,B 0,C 180,E1 -12672.849,E2 -12672.849} C_VEL
LIN {X 0,Y 371.036,Z 785.073,A -85,B 0,C 180,E1 -12674.059,E2 -12674.059} C_VEL
LIN {X 0,Y 370.035,Z 796.366,A -85,B 0,C 180,E1 -12675.425,E2 -12675.425} C_VEL
LIN {X 0,Y 369.044,Z 809.203,A -85,B 0,C 180,E1 -12677.35,E2 -12677.35} C_VEL
LIN {X 0,Y 368.459,Z 818.314,A -85,B 0,C 180,E1 -12679.005,E2 -12679.005} C_VEL
LIN {X 0,Y 368.19,Z 825.705,A -85,B 0,C 180,E1 -12680.663,E2 -12680.663} C_VEL
LIN {X 0,Y 368.117,Z 831.592,A -85,B 0,C 180,E1 -12682.321,E2 -12682.321} C_VEL
LIN {X 0,Y 368.181,Z 836.19,A -85,B 0,C 180,E1 -12683.974,E2 -12683.974} C_VEL
LIN {X 0,Y 368.412,Z 839.635,A -85,B 0,C 180,E1 -12685.624,E2 -12685.624} C_VEL
LIN {X 0,Y 368.392,Z 841.26,A -85,B 0,C 180,E1 -12686.72,E2 -12686.72} C_VEL
LIN {X 0,Y 368.42,Z 842.435,A -85,B 0,C 180,E1 -12687.814,E2 -12687.814} C_VEL
LIN {X 0,Y 368.507,Z 843.171,A -85,B 0,C 180,E1 -12688.908,E2 -12688.908} C_VEL
LIN {X 0,Y 368.699,Z 843.446,A -85,B 0,C 180,E1 -12690.001,E2 -12690.001} C_VEL
LIN {X 0,Y 368.455,Z 843.175,A -85,B 0,C 180,E1 -12691.094,E2 -12691.094} C_VEL
LIN {X 0,Y 368.4,Z 842.494,A -85,B 0,C 180,E1 -12692.187,E2 -12692.187} C_VEL
LIN {X 0,Y 368.367,Z 841.37,A -85,B 0,C 180,E1 -12693.282,E2 -12693.282} C_VEL
LIN {X 0,Y 368.276,Z 838.783,A -85,B 0,C 180,E1 -12694.927,E2 -12694.927} C_VEL
LIN {X 0,Y 368.105,Z 834.363,A -85,B 0,C 180,E1 -12696.874,E2 -12696.874} C_VEL
LIN {X 0,Y 368.088,Z 828.443,A -85,B 0,C 180,E1 -12698.787,E2 -12698.787} C_VEL
LIN {X 0,Y 368.293,Z 820.734,A -85,B 0,C 180,E1 -12700.723,E2 -12700.723} C_VEL
LIN {X 0,Y 368.828,Z 812.55,A -85,B 0,C 180,E1 -12702.379,E2 -12702.379} C_VEL
LIN {X 0,Y 369.33,Z 804.123,A -85,B 0,C 180,E1 -12703.8,E2 -12703.8} C_VEL
LIN {X 0,Y 370.407,Z 794.709,A -85,B 0,C 180,E1 -12705.123,E2 -12705.123} C_VEL
LIN {X 0,Y 371.5,Z 784.367,A -85,B 0,C 180,E1 -12706.345,E2 -12706.345} C_VEL
LIN {X 0,Y 372.933,Z 771.865,A -85,B 0,C 180,E1 -12707.55,E2 -12707.55} C_VEL
LIN {X 0,Y 374.413,Z 758.171,A -85,B 0,C 180,E1 -12708.609,E2 -12708.609} C_VEL
LIN {X 0,Y 375.906,Z 743.877,A -85,B 0,C 180,E1 -12709.453,E2 -12709.453} C_VEL
LIN {X 0,Y 377.122,Z 728.396,A -85,B 0,C 180,E1 -12710.132,E2 -12710.132} C_VEL
LIN {X 0,Y 378.03,Z 709.508,A -85,B 0,C 180,E1 -12710.686,E2 -12710.686} C_VEL
LIN {X 0,Y 379.111,Z 677.459,A -85,B 0,C 180,E1 -12711.546,E2 -12711.546} C_VEL
LIN {X 0,Y 377.52,Z 643.927,A -85,B 0,C 180,E1 -12712.739,E2 -12712.739} C_VEL
LIN {X 0,Y 375.525,Z 624.714,A -85,B 0,C 180,E1 -12713.568,E2 -12713.568} C_VEL
LIN {X 0,Y 372.6,Z 606.71,A -85,B 0,C 180,E1 -12714.506,E2 -12714.506} C_VEL
LIN {X 0,Y 370.481,Z 595.909,A -85,B 0,C 180,E1 -12715.133,E2 -12715.133} C_VEL
LIN {X 0,Y 369.569,Z 590.784,A -85,B 0,C 180,E1 -12715.446,E2 -12715.446} C_VEL
LIN {X 0,Y 370.385,Z 573.335,A -85,B 0,C 180,E1 -12719.209,E2 -12719.209} C_VEL
LIN {X 0,Y 370.77,Z 564.86,A -85,B 0,C 180,E1 -12721.106,E2 -12721.106} C_VEL
LIN {X 0,Y 369.643,Z 557.977,A -85,B 0,C 180,E1 -12722.779,E2 -12722.779} C_VEL
LIN {X 0,Y 368.999,Z 554.524,A -85,B 0,C 180,E1 -12723.692,E2 -12723.692} C_VEL
LIN {X 0,Y 368.908,Z 554.531,A -85,B 0,C 180,E1 -12727.563,E2 -12727.563} C_VEL
LIN {X 0,Y 368.915,Z 554.529,A -85,B 0,C 180,E1 -12730.37,E2 -12730.37} C_VEL
LIN {X 0,Y 368.887,Z 554.534,A -85,B 0,C 180,E1 -12733.616,E2 -12733.616} C_VEL
LIN {X 0,Y 368.89,Z 554.533,A -85,B 0,C 180,E1 -12736.696,E2 -12736.696} C_VEL
LIN {X 0,Y 368.916,Z 554.531,A -85,B 0,C 180,E1 -12739.643,E2 -12739.643} C_VEL
LIN {X 0,Y 368.906,Z 554.534,A -85,B 0,C 180,E1 -12743.144,E2 -12743.144} C_VEL
LIN {X 0,Y 368.901,Z 554.532,A -85,B 0,C 180,E1 -12746.462,E2 -12746.462} C_VEL
LIN {X 0,Y 368.934,Z 554.53,A -85,B 0,C 180,E1 -12749.046,E2 -12749.046} C_VEL
LIN {X 0,Y 368.968,Z 554.527,A -85,B 0,C 180,E1 -12752.796,E2 -12752.796} C_VEL
LIN {X 0,Y 368.979,Z 554.527,A -85,B 0,C 180,E1 -12754.559,E2 -12754.559} C_VEL
LIN {X 0,Y 369.983,Z 557.393,A -85,B 0,C 180,E1 -12754.775,E2 -12754.775} C_VEL
LIN {X 0,Y 371.653,Z 559.764,A -85,B 0,C 180,E1 -12755.052,E2 -12755.052} C_VEL
LIN {X 0,Y 378.013,Z 570.939,A -85,B 0,C 180,E1 -12756.082,E2 -12756.082} C_VEL
LIN {X 0,Y 382.715,Z 580.791,A -85,B 0,C 180,E1 -12756.828,E2 -12756.828} C_VEL
LIN {X 0,Y 382.596,Z 612.183,A -85,B 0,C 180,E1 -12757.605,E2 -12757.605} C_VEL
LIN {X 0,Y 382.423,Z 626.755,A -85,B 0,C 180,E1 -12758.167,E2 -12758.167} C_VEL
LIN {X 0,Y 381.911,Z 640.464,A -85,B 0,C 180,E1 -12758.9,E2 -12758.9} C_VEL
LIN {X 0,Y 380.997,Z 655.371,A -85,B 0,C 180,E1 -12759.948,E2 -12759.948} C_VEL
LIN {X 0,Y 379.98,Z 668.071,A -85,B 0,C 180,E1 -12761.081,E2 -12761.081} C_VEL
LIN {X 0,Y 378.801,Z 679.382,A -85,B 0,C 180,E1 -12762.313,E2 -12762.313} C_VEL
LIN {X 0,Y 377.467,Z 690.469,A -85,B 0,C 180,E1 -12763.782,E2 -12763.782} C_VEL
LIN {X 0,Y 376.102,Z 700.51,A -85,B 0,C 180,E1 -12765.388,E2 -12765.388} C_VEL
LIN {X 0,Y 374.857,Z 708.889,A -85,B 0,C 180,E1 -12766.998,E2 -12766.998} C_VEL
LIN {X 0,Y 373.568,Z 716.958,A -85,B 0,C 180,E1 -12768.881,E2 -12768.881} C_VEL
LIN {X 0,Y 372.445,Z 723.515,A -85,B 0,C 180,E1 -12770.77,E2 -12770.77} C_VEL
LIN {X 0,Y 371.514,Z 728.162,A -85,B 0,C 180,E1 -12772.39,E2 -12772.39} C_VEL
LIN {X 0,Y 370.978,Z 731.844,A -85,B 0,C 180,E1 -12774.019,E2 -12774.019} C_VEL
LIN {X 0,Y 370.449,Z 734.801,A -85,B 0,C 180,E1 -12775.647,E2 -12775.647} C_VEL
LIN {X 0,Y 369.842,Z 737.566,A -85,B 0,C 180,E1 -12777.821,E2 -12777.821} C_VEL
LIN {X 0,Y 369.443,Z 739.07,A -85,B 0,C 180,E1 -12780,E2 -12780} C_VEL
LIN {X 0,Y 369.206,Z 739.338,A -85,B 0,C 180,E1 -12782.181,E2 -12782.181} C_VEL
LIN {X 0,Y 368.972,Z 738.392,A -85,B 0,C 180,E1 -12784.369,E2 -12784.369} C_VEL
LIN {X 0,Y 369.299,Z 736.097,A -85,B 0,C 180,E1 -12786.596,E2 -12786.596} C_VEL
LIN {X 0,Y 369.347,Z 732.685,A -85,B 0,C 180,E1 -12788.755,E2 -12788.755} C_VEL
LIN {X 0,Y 369.655,Z 727.834,A -85,B 0,C 180,E1 -12790.959,E2 -12790.959} C_VEL
LIN {X 0,Y 370.099,Z 721.471,A -85,B 0,C 180,E1 -12793.171,E2 -12793.171} C_VEL
LIN {X 0,Y 370.636,Z 715.33,A -85,B 0,C 180,E1 -12794.887,E2 -12794.887} C_VEL
LIN {X 0,Y 371.412,Z 707.246,A -85,B 0,C 180,E1 -12796.772,E2 -12796.772} C_VEL
LIN {X 0,Y 372.189,Z 698.711,A -85,B 0,C 180,E1 -12798.438,E2 -12798.438} C_VEL
LIN {X 0,Y 373.094,Z 688.57,A -85,B 0,C 180,E1 -12800.107,E2 -12800.107} C_VEL
LIN {X 0,Y 374.047,Z 677.464,A -85,B 0,C 180,E1 -12801.637,E2 -12801.637} C_VEL
LIN {X 0,Y 375.057,Z 665.371,A -85,B 0,C 180,E1 -12803.026,E2 -12803.026} C_VEL
LIN {X 0,Y 375.921,Z 652.141,A -85,B 0,C 180,E1 -12804.286,E2 -12804.286} C_VEL
LIN {X 0,Y 376.668,Z 639.501,A -85,B 0,C 180,E1 -12805.265,E2 -12805.265} C_VEL
LIN {X 0,Y 377.374,Z 624.673,A -85,B 0,C 180,E1 -12806.176,E2 -12806.176} C_VEL
LIN {X 0,Y 377.867,Z 610.041,A -85,B 0,C 180,E1 -12806.852,E2 -12806.852} C_VEL
LIN {X 0,Y 378.033,Z 595.276,A -85,B 0,C 180,E1 -12807.333,E2 -12807.333} C_VEL
LIN {X 0,Y 378.093,Z 579.25,A -85,B 0,C 180,E1 -12807.721,E2 -12807.721} C_VEL
LIN {X 0,Y 368.934,Z 554.528,A -85,B 0,C 180,E1 -12808.803,E2 -12808.803} C_VEL
LIN {X 0,Y 368.899,Z 554.534,A -85,B 0,C 180,E1 -12812.237,E2 -12812.237} C_VEL
LIN {X 0,Y 368.93,Z 554.525,A -85,B 0,C 180,E1 -12815.001,E2 -12815.001} C_VEL
LIN {X 0,Y 368.909,Z 554.53,A -85,B 0,C 180,E1 -12818.639,E2 -12818.639} C_VEL
LIN {X 0,Y 368.882,Z 554.535,A -85,B 0,C 180,E1 -12822.009,E2 -12822.009} C_VEL
LIN {X 0,Y 368.88,Z 554.532,A -85,B 0,C 180,E1 -12825.175,E2 -12825.175} C_VEL
LIN {X 0,Y 368.883,Z 554.536,A -85,B 0,C 180,E1 -12828.177,E2 -12828.177} C_VEL
LIN {X 0,Y 368.91,Z 554.528,A -85,B 0,C 180,E1 -12831.359,E2 -12831.359} C_VEL
LIN {X 0,Y 368.936,Z 554.526,A -85,B 0,C 180,E1 -12835.146,E2 -12835.146} C_VEL
LIN {X 0,Y 368.928,Z 554.528,A -85,B 0,C 180,E1 -12839.046,E2 -12839.046} C_VEL
LIN {X 0,Y 368.962,Z 554.527,A -85,B 0,C 180,E1 -12842.796,E2 -12842.796} C_VEL
LIN {X 0,Y 368.944,Z 554.525,A -85,B 0,C 180,E1 -12846.112,E2 -12846.112} C_VEL
LIN {X 0,Y 368.935,Z 554.525,A -85,B 0,C 180,E1 -12849.946,E2 -12849.946} C_VEL
LIN {X 0,Y 368.974,Z 554.521,A -85,B 0,C 180,E1 -12853.398,E2 -12853.398} C_VEL
LIN {X 0,Y 369.056,Z 554.515,A -85,B 0,C 180,E1 -12856.79,E2 -12856.79} C_VEL
LIN {X 0,Y 369.066,Z 554.509,A -85,B 0,C 180,E1 -12860.131,E2 -12860.131} C_VEL
LIN {X 0,Y 369.186,Z 554.494,A -85,B 0,C 180,E1 -12862.342,E2 -12862.342} C_VEL
LIN {X 0,Y 369.143,Z 554.501,A -85,B 0,C 180,E1 -12864.537,E2 -12864.537} C_VEL
LIN {X 0,Y 369.317,Z 554.478,A -85,B 0,C 180,E1 -12867.818,E2 -12867.818} C_VEL
LIN {X 0,Y 369.456,Z 554.46,A -85,B 0,C 180,E1 -12869.999,E2 -12869.999} C_VEL
LIN {X 0,Y 369.317,Z 554.477,A -85,B 0,C 180,E1 -12872.181,E2 -12872.181} C_VEL
LIN {X 0,Y 369.203,Z 554.492,A -85,B 0,C 180,E1 -12876.558,E2 -12876.558} C_VEL
LIN {X 0,Y 369.135,Z 554.501,A -85,B 0,C 180,E1 -12878.76,E2 -12878.76} C_VEL
LIN {X 0,Y 369.011,Z 554.516,A -85,B 0,C 180,E1 -12882.092,E2 -12882.092} C_VEL
LIN {X 0,Y 368.995,Z 554.524,A -85,B 0,C 180,E1 -12885.464,E2 -12885.464} C_VEL
LIN {X 0,Y 368.954,Z 554.523,A -85,B 0,C 180,E1 -12888.894,E2 -12888.894} C_VEL
LIN {X 0,Y 368.931,Z 554.525,A -85,B 0,C 180,E1 -12892.394,E2 -12892.394} C_VEL
LIN {X 0,Y 368.996,Z 554.52,A -85,B 0,C 180,E1 -12895.98,E2 -12895.98} C_VEL
LIN {X 0,Y 368.965,Z 554.521,A -85,B 0,C 180,E1 -12898.814,E2 -12898.814} C_VEL
LIN {X 0,Y 368.906,Z 554.53,A -85,B 0,C 180,E1 -12902.236,E2 -12902.236} C_VEL
LIN {X 0,Y 368.905,Z 554.527,A -85,B 0,C 180,E1 -12905.331,E2 -12905.331} C_VEL
LIN {X 0,Y 368.225,Z 554.616,A -85,B 0,C 180,E1 -12906.243,E2 -12906.243} C_VEL
LIN {X 0,Y 365.383,Z 554.974,A -85,B 0,C 180,E1 -12907.726,E2 -12907.726} C_VEL
LIN {X 0,Y 362.984,Z 555.275,A -85,B 0,C 180,E1 -12908.925,E2 -12908.925} C_VEL
LIN {X 0,Y 361.949,Z 555.402,A -85,B 0,C 180,E1 -12909.853,E2 -12909.853} C_VEL
LIN {X 0,Y 361.862,Z 555.409,A -85,B 0,C 180,E1 -12910.167,E2 -12910.167} C_VEL
LIN {X 0,Y 361.855,Z 555.412,A -85,B 0,C 180,E1 -12914.06,E2 -12914.06} C_VEL
LIN {X 0,Y 361.88,Z 555.404,A -85,B 0,C 180,E1 -12917.178,E2 -12917.178} C_VEL
LIN {X 0,Y 361.875,Z 555.41,A -85,B 0,C 180,E1 -12920.142,E2 -12920.142} C_VEL
LIN {X 0,Y 361.887,Z 555.404,A -85,B 0,C 180,E1 -12923.494,E2 -12923.494} C_VEL
LIN {X 0,Y 370.245,Z 578.188,A -85,B 0,C 180,E1 -12924.475,E2 -12924.475} C_VEL
LIN {X 0,Y 369.594,Z 615.713,A -85,B 0,C 180,E1 -12925.357,E2 -12925.357} C_VEL
LIN {X 0,Y 369.38,Z 630.513,A -85,B 0,C 180,E1 -12925.918,E2 -12925.918} C_VEL
LIN {X 0,Y 368.858,Z 644.082,A -85,B 0,C 180,E1 -12926.646,E2 -12926.646} C_VEL
LIN {X 0,Y 368.142,Z 657.269,A -85,B 0,C 180,E1 -12927.583,E2 -12927.583} C_VEL
LIN {X 0,Y 367.337,Z 670.048,A -85,B 0,C 180,E1 -12928.738,E2 -12928.738} C_VEL
LIN {X 0,Y 366.38,Z 682.11,A -85,B 0,C 180,E1 -12930.084,E2 -12930.084} C_VEL
LIN {X 0,Y 365.519,Z 693.018,A -85,B 0,C 180,E1 -12931.578,E2 -12931.578} C_VEL
LIN {X 0,Y 364.721,Z 702.063,A -85,B 0,C 180,E1 -12933.075,E2 -12933.075} C_VEL
LIN {X 0,Y 363.919,Z 710.955,A -85,B 0,C 180,E1 -12934.859,E2 -12934.859} C_VEL
LIN {X 0,Y 363.239,Z 718.216,A -85,B 0,C 180,E1 -12936.632,E2 -12936.632} C_VEL
LIN {X 0,Y 362.696,Z 724.266,A -85,B 0,C 180,E1 -12938.448,E2 -12938.448} C_VEL
LIN {X 0,Y 362.353,Z 728.849,A -85,B 0,C 180,E1 -12940.159,E2 -12940.159} C_VEL
LIN {X 0,Y 362.083,Z 732.694,A -85,B 0,C 180,E1 -12942.002,E2 -12942.002} C_VEL
LIN {X 0,Y 361.838,Z 735.935,A -85,B 0,C 180,E1 -12944.222,E2 -12944.222} C_VEL
LIN {X 0,Y 361.914,Z 737.81,A -85,B 0,C 180,E1 -12946.525,E2 -12946.525} C_VEL
LIN {X 0,Y 361.944,Z 738.201,A -85,B 0,C 180,E1 -12947.668,E2 -12947.668} C_VEL
LIN {X 0,Y 362.203,Z 737.815,A -85,B 0,C 180,E1 -12949.943,E2 -12949.943} C_VEL
LIN {X 0,Y 362.629,Z 735.985,A -85,B 0,C 180,E1 -12952.203,E2 -12952.203} C_VEL
LIN {X 0,Y 363.263,Z 732.704,A -85,B 0,C 180,E1 -12954.449,E2 -12954.449} C_VEL
LIN {X 0,Y 363.835,Z 729.192,A -85,B 0,C 180,E1 -12956.124,E2 -12956.124} C_VEL
LIN {X 0,Y 364.588,Z 724.728,A -85,B 0,C 180,E1 -12957.791,E2 -12957.791} C_VEL
LIN {X 0,Y 365.598,Z 718.295,A -85,B 0,C 180,E1 -12959.697,E2 -12959.697} C_VEL
LIN {X 0,Y 366.642,Z 711.242,A -85,B 0,C 180,E1 -12961.373,E2 -12961.373} C_VEL
LIN {X 0,Y 367.849,Z 702.802,A -85,B 0,C 180,E1 -12963.012,E2 -12963.012} C_VEL
LIN {X 0,Y 368.861,Z 694.436,A -85,B 0,C 180,E1 -12964.371,E2 -12964.371} C_VEL
LIN {X 0,Y 370.055,Z 684.384,A -85,B 0,C 180,E1 -12965.723,E2 -12965.723} C_VEL
LIN {X 0,Y 371.13,Z 673.394,A -85,B 0,C 180,E1 -12966.934,E2 -12966.934} C_VEL
LIN {X 0,Y 372.194,Z 661.154,A -85,B 0,C 180,E1 -12968.005,E2 -12968.005} C_VEL
LIN {X 0,Y 372.908,Z 647.55,A -85,B 0,C 180,E1 -12968.945,E2 -12968.945} C_VEL
LIN {X 0,Y 373.408,Z 633.642,A -85,B 0,C 180,E1 -12969.65,E2 -12969.65} C_VEL
LIN {X 0,Y 373.521,Z 619.334,A -85,B 0,C 180,E1 -12970.146,E2 -12970.146} C_VEL
LIN {X 0,Y 374.279,Z 582.841,A -85,B 0,C 180,E1 -12971.012,E2 -12971.012} C_VEL
LIN {X 0,Y 374.203,Z 579.864,A -85,B 0,C 180,E1 -12971.096,E2 -12971.096} C_VEL
LIN {X 0,Y 368.213,Z 567.528,A -85,B 0,C 180,E1 -12972.004,E2 -12972.004} C_VEL
LIN {X 0,Y 363.224,Z 558.545,A -85,B 0,C 180,E1 -12972.784,E2 -12972.784} C_VEL
LIN {X 0,Y 362.093,Z 555.832,A -85,B 0,C 180,E1 -12972.987,E2 -12972.987} C_VEL
LIN {X 0,Y 362.011,Z 555.397,A -85,B 0,C 180,E1 -12973.043,E2 -12973.043} C_VEL
LIN {X 0,Y 361.93,Z 555.405,A -85,B 0,C 180,E1 -12976.935,E2 -12976.935} C_VEL
LIN {X 0,Y 361.891,Z 555.407,A -85,B 0,C 180,E1 -12980.461,E2 -12980.461} C_VEL
LIN {X 0,Y 361.893,Z 555.406,A -85,B 0,C 180,E1 -12984.114,E2 -12984.114} C_VEL
LIN {X 0,Y 361.94,Z 555.398,A -85,B 0,C 180,E1 -12986.723,E2 -12986.723} C_VEL
LIN {X 0,Y 361.874,Z 555.4,A -85,B 0,C 180,E1 -12990.329,E2 -12990.329} C_VEL
LIN {X 0,Y 361.852,Z 555.402,A -85,B 0,C 180,E1 -12994.281,E2 -12994.281} C_VEL
LIN {X 0,Y 361.863,Z 555.403,A -85,B 0,C 180,E1 -12997.224,E2 -12997.224} C_VEL
LIN {X 0,Y 361.835,Z 555.412,A -85,B 0,C 180,E1 -13000.757,E2 -13000.757} C_VEL
LIN {X 0,Y 361.82,Z 555.412,A -85,B 0,C 180,E1 -13004.369,E2 -13004.369} C_VEL
LIN {X 0,Y 361.835,Z 555.412,A -85,B 0,C 180,E1 -13007.569,E2 -13007.569} C_VEL
LIN {X 0,Y 361.934,Z 555.5,A -85,B 0,C 180,E1 -13011.508,E2 -13011.508} C_VEL
LIN {X 0,Y 364.884,Z 569.98,A -85,B 0,C 180,E1 -13015.302,E2 -13015.302} C_VEL
LIN {X 0,Y 366.752,Z 578.885,A -85,B 0,C 180,E1 -13017.551,E2 -13017.551} C_VEL
LIN {X 0,Y 365.447,Z 592.145,A -85,B 0,C 180,E1 -13020.634,E2 -13020.634} C_VEL
LIN {X 0,Y 363.918,Z 609.207,A -85,B 0,C 180,E1 -13024.553,E2 -13024.553} C_VEL
LIN {X 0,Y 363.431,Z 615.903,A -85,B 0,C 180,E1 -13026.08,E2 -13026.08} C_VEL
LIN {X 0,Y 364.113,Z 620.421,A -85,B 0,C 180,E1 -13026.294,E2 -13026.294} C_VEL
LIN {X 0,Y 366.76,Z 637.153,A -85,B 0,C 180,E1 -13027.072,E2 -13027.072} C_VEL
LIN {X 0,Y 370.977,Z 678.992,A -85,B 0,C 180,E1 -13028.682,E2 -13028.682} C_VEL
LIN {X 0,Y 369.302,Z 729.569,A -85,B 0,C 180,E1 -13030.005,E2 -13030.005} C_VEL
LIN {X 0,Y 368.436,Z 743.498,A -85,B 0,C 180,E1 -13030.573,E2 -13030.573} C_VEL
LIN {X 0,Y 367.266,Z 756.477,A -85,B 0,C 180,E1 -13031.306,E2 -13031.306} C_VEL
LIN {X 0,Y 365.925,Z 769.216,A -85,B 0,C 180,E1 -13032.249,E2 -13032.249} C_VEL
LIN {X 0,Y 364.667,Z 780.923,A -85,B 0,C 180,E1 -13033.342,E2 -13033.342} C_VEL
LIN {X 0,Y 363.54,Z 791.647,A -85,B 0,C 180,E1 -13034.585,E2 -13034.585} C_VEL
LIN {X 0,Y 362.525,Z 802.375,A -85,B 0,C 180,E1 -13036.116,E2 -13036.116} C_VEL
LIN {X 0,Y 361.834,Z 811.267,A -85,B 0,C 180,E1 -13037.664,E2 -13037.664} C_VEL
LIN {X 0,Y 361.2,Z 821.942,A -85,B 0,C 180,E1 -13039.915,E2 -13039.915} C_VEL
LIN {X 0,Y 361.099,Z 828.391,A -85,B 0,C 180,E1 -13041.607,E2 -13041.607} C_VEL
LIN {X 0,Y 361.088,Z 833.476,A -85,B 0,C 180,E1 -13043.294,E2 -13043.294} C_VEL
LIN {X 0,Y 361.327,Z 837.372,A -85,B 0,C 180,E1 -13044.979,E2 -13044.979} C_VEL
LIN {X 0,Y 361.366,Z 840.096,A -85,B 0,C 180,E1 -13046.656,E2 -13046.656} C_VEL
LIN {X 0,Y 361.397,Z 841.299,A -85,B 0,C 180,E1 -13047.772,E2 -13047.772} C_VEL
LIN {X 0,Y 361.503,Z 842.061,A -85,B 0,C 180,E1 -13048.887,E2 -13048.887} C_VEL
LIN {X 0,Y 361.699,Z 842.384,A -85,B 0,C 180,E1 -13050.001,E2 -13050.001} C_VEL
LIN {X 0,Y 361.423,Z 842.141,A -85,B 0,C 180,E1 -13051.115,E2 -13051.115} C_VEL
LIN {X 0,Y 361.36,Z 841.473,A -85,B 0,C 180,E1 -13052.23,E2 -13052.23} C_VEL
LIN {X 0,Y 361.319,Z 840.37,A -85,B 0,C 180,E1 -13053.346,E2 -13053.346} C_VEL
LIN {X 0,Y 361.209,Z 837.825,A -85,B 0,C 180,E1 -13055.024,E2 -13055.024} C_VEL
LIN {X 0,Y 361.039,Z 833.74,A -85,B 0,C 180,E1 -13056.891,E2 -13056.891} C_VEL
LIN {X 0,Y 360.981,Z 829.444,A -85,B 0,C 180,E1 -13058.397,E2 -13058.397} C_VEL
LIN {X 0,Y 361.133,Z 822.338,A -85,B 0,C 180,E1 -13060.371,E2 -13060.371} C_VEL
LIN {X 0,Y 361.634,Z 814.774,A -85,B 0,C 180,E1 -13062.059,E2 -13062.059} C_VEL
LIN {X 0,Y 362.24,Z 805.856,A -85,B 0,C 180,E1 -13063.694,E2 -13063.694} C_VEL
LIN {X 0,Y 363.407,Z 795.307,A -85,B 0,C 180,E1 -13065.278,E2 -13065.278} C_VEL
LIN {X 0,Y 364.538,Z 785.34,A -85,B 0,C 180,E1 -13066.522,E2 -13066.522} C_VEL
LIN {X 0,Y 366.003,Z 773.472,A -85,B 0,C 180,E1 -13067.749,E2 -13067.749} C_VEL
LIN {X 0,Y 367.521,Z 760.542,A -85,B 0,C 180,E1 -13068.827,E2 -13068.827} C_VEL
LIN {X 0,Y 369.289,Z 745.209,A -85,B 0,C 180,E1 -13069.816,E2 -13069.816} C_VEL
LIN {X 0,Y 370.61,Z 730.117,A -85,B 0,C 180,E1 -13070.538,E2 -13070.538} C_VEL
LIN {X 0,Y 371.584,Z 713.956,A -85,B 0,C 180,E1 -13071.082,E2 -13071.082} C_VEL
LIN {X 0,Y 372.924,Z 678,A -85,B 0,C 180,E1 -13072.077,E2 -13072.077} C_VEL
LIN {X 0,Y 371.533,Z 645.199,A -85,B 0,C 180,E1 -13073.285,E2 -13073.285} C_VEL
LIN {X 0,Y 369.562,Z 625.703,A -85,B 0,C 180,E1 -13074.165,E2 -13074.165} C_VEL
LIN {X 0,Y 366.886,Z 608.736,A -85,B 0,C 180,E1 -13075.082,E2 -13075.082} C_VEL
LIN {X 0,Y 364.837,Z 598.041,A -85,B 0,C 180,E1 -13075.735,E2 -13075.735} C_VEL
LIN {X 0,Y 363.58,Z 592.147,A -85,B 0,C 180,E1 -13076.129,E2 -13076.129} C_VEL
LIN {X 0,Y 362.696,Z 587.099,A -85,B 0,C 180,E1 -13076.467,E2 -13076.467} C_VEL
LIN {X 0,Y 363.611,Z 570.513,A -85,B 0,C 180,E1 -13080.169,E2 -13080.169} C_VEL
LIN {X 0,Y 363.735,Z 565.036,A -85,B 0,C 180,E1 -13081.446,E2 -13081.446} C_VEL
LIN {X 0,Y 361.932,Z 555.404,A -85,B 0,C 180,E1 -13083.925,E2 -13083.925} C_VEL
LIN {X 0,Y 361.868,Z 555.411,A -85,B 0,C 180,E1 -13087.223,E2 -13087.223} C_VEL
LIN {X 0,Y 361.84,Z 555.412,A -85,B 0,C 180,E1 -13090.755,E2 -13090.755} C_VEL
LIN {X 0,Y 361.821,Z 555.412,A -85,B 0,C 180,E1 -13094.369,E2 -13094.369} C_VEL
LIN {X 0,Y 361.84,Z 555.413,A -85,B 0,C 180,E1 -13097.568,E2 -13097.568} C_VEL
LIN {X 0,Y 361.875,Z 555.408,A -85,B 0,C 180,E1 -13100.973,E2 -13100.973} C_VEL
LIN {X 0,Y 361.879,Z 555.407,A -85,B 0,C 180,E1 -13104.655,E2 -13104.655} C_VEL
LIN {X 0,Y 361.842,Z 555.412,A -85,B 0,C 180,E1 -13108.37,E2 -13108.37} C_VEL
LIN {X 0,Y 361.913,Z 555.409,A -85,B 0,C 180,E1 -13112.221,E2 -13112.221} C_VEL
LIN {X 0,Y 361.967,Z 555.402,A -85,B 0,C 180,E1 -13113.641,E2 -13113.641} C_VEL
LIN {X 0,Y 362.952,Z 558.249,A -85,B 0,C 180,E1 -13113.879,E2 -13113.879} C_VEL
LIN {X 0,Y 364.771,Z 560.778,A -85,B 0,C 180,E1 -13114.213,E2 -13114.213} C_VEL
LIN {X 0,Y 371.321,Z 571.921,A -85,B 0,C 180,E1 -13115.362,E2 -13115.362} C_VEL
LIN {X 0,Y 376.873,Z 583.156,A -85,B 0,C 180,E1 -13116.281,E2 -13116.281} C_VEL
LIN {X 0,Y 376.575,Z 612.609,A -85,B 0,C 180,E1 -13117.039,E2 -13117.039} C_VEL
LIN {X 0,Y 376.414,Z 627.29,A -85,B 0,C 180,E1 -13117.596,E2 -13117.596} C_VEL
LIN {X 0,Y 375.922,Z 641.119,A -85,B 0,C 180,E1 -13118.331,E2 -13118.331} C_VEL
LIN {X 0,Y 375.04,Z 655.167,A -85,B 0,C 180,E1 -13119.316,E2 -13119.316} C_VEL
LIN {X 0,Y 373.992,Z 667.315,A -85,B 0,C 180,E1 -13120.385,E2 -13120.385} C_VEL
LIN {X 0,Y 372.679,Z 679.701,A -85,B 0,C 180,E1 -13121.728,E2 -13121.728} C_VEL
LIN {X 0,Y 371.52,Z 689.151,A -85,B 0,C 180,E1 -13122.949,E2 -13122.949} C_VEL
LIN {X 0,Y 370.015,Z 699.628,A -85,B 0,C 180,E1 -13124.578,E2 -13124.578} C_VEL
LIN {X 0,Y 368.65,Z 708.335,A -85,B 0,C 180,E1 -13126.213,E2 -13126.213} C_VEL
LIN {X 0,Y 367.224,Z 716.719,A -85,B 0,C 180,E1 -13128.127,E2 -13128.127} C_VEL
LIN {X 0,Y 365.99,Z 723.58,A -85,B 0,C 180,E1 -13130.047,E2 -13130.047} C_VEL
LIN {X 0,Y 364.682,Z 729.789,A -85,B 0,C 180,E1 -13132.247,E2 -13132.247} C_VEL
LIN {X 0,Y 364.109,Z 733.382,A -85,B 0,C 180,E1 -13133.905,E2 -13133.905} C_VEL
LIN {X 0,Y 363.512,Z 736.215,A -85,B 0,C 180,E1 -13135.564,E2 -13135.564} C_VEL
LIN {X 0,Y 362.872,Z 738.873,A -85,B 0,C 180,E1 -13137.78,E2 -13137.78} C_VEL
LIN {X 0,Y 362.459,Z 740.263,A -85,B 0,C 180,E1 -13140,E2 -13140} C_VEL
LIN {X 0,Y 362.186,Z 740.42,A -85,B 0,C 180,E1 -13142.224,E2 -13142.224} C_VEL
LIN {X 0,Y 361.95,Z 739.357,A -85,B 0,C 180,E1 -13144.454,E2 -13144.454} C_VEL
LIN {X 0,Y 362.276,Z 737,A -85,B 0,C 180,E1 -13146.684,E2 -13146.684} C_VEL
LIN {X 0,Y 362.35,Z 733.392,A -85,B 0,C 180,E1 -13148.926,E2 -13148.926} C_VEL
LIN {X 0,Y 362.676,Z 728.379,A -85,B 0,C 180,E1 -13151.173,E2 -13151.173} C_VEL
LIN {X 0,Y 363.151,Z 721.825,A -85,B 0,C 180,E1 -13153.428,E2 -13153.428} C_VEL
LIN {X 0,Y 363.798,Z 714.679,A -85,B 0,C 180,E1 -13155.401,E2 -13155.401} C_VEL
LIN {X 0,Y 364.654,Z 705.926,A -85,B 0,C 180,E1 -13157.381,E2 -13157.381} C_VEL
LIN {X 0,Y 365.627,Z 695.707,A -85,B 0,C 180,E1 -13159.288,E2 -13159.288} C_VEL
LIN {X 0,Y 366.631,Z 684.21,A -85,B 0,C 180,E1 -13161.064,E2 -13161.064} C_VEL
LIN {X 0,Y 367.651,Z 671.992,A -85,B 0,C 180,E1 -13162.625,E2 -13162.625} C_VEL
LIN {X 0,Y 368.56,Z 659.939,A -85,B 0,C 180,E1 -13163.903,E2 -13163.903} C_VEL
LIN {X 0,Y 369.48,Z 646.941,A -85,B 0,C 180,E1 -13165.038,E2 -13165.038} C_VEL
LIN {X 0,Y 370.255,Z 632.729,A -85,B 0,C 180,E1 -13166.036,E2 -13166.036} C_VEL
LIN {X 0,Y 370.896,Z 617.534,A -85,B 0,C 180,E1 -13166.856,E2 -13166.856} C_VEL
LIN {X 0,Y 371.175,Z 601.94,A -85,B 0,C 180,E1 -13167.465,E2 -13167.465} C_VEL
LIN {X 0,Y 371.301,Z 580.779,A -85,B 0,C 180,E1 -13168.012,E2 -13168.012} C_VEL
LIN {X 0,Y 361.884,Z 555.416,A -85,B 0,C 180,E1 -13169.127,E2 -13169.127} C_VEL
LIN {X 0,Y 361.85,Z 555.408,A -85,B 0,C 180,E1 -13172.944,E2 -13172.944} C_VEL
LIN {X 0,Y 361.869,Z 555.407,A -85,B 0,C 180,E1 -13175.636,E2 -13175.636} C_VEL
LIN {X 0,Y 361.87,Z 555.405,A -85,B 0,C 180,E1 -13179.026,E2 -13179.026} C_VEL
LIN {X 0,Y 361.836,Z 555.411,A -85,B 0,C 180,E1 -13182.828,E2 -13182.828} C_VEL
LIN {X 0,Y 361.818,Z 555.414,A -85,B 0,C 180,E1 -13185.946,E2 -13185.946} C_VEL
LIN {X 0,Y 361.836,Z 555.409,A -85,B 0,C 180,E1 -13189.244,E2 -13189.244} C_VEL
LIN {X 0,Y 361.871,Z 555.408,A -85,B 0,C 180,E1 -13192.775,E2 -13192.775} C_VEL
LIN {X 0,Y 361.854,Z 555.407,A -85,B 0,C 180,E1 -13195.719,E2 -13195.719} C_VEL
LIN {X 0,Y 361.872,Z 555.405,A -85,B 0,C 180,E1 -13199.671,E2 -13199.671} C_VEL
LIN {X 0,Y 361.953,Z 555.395,A -85,B 0,C 180,E1 -13203.474,E2 -13203.474} C_VEL
LIN {X 0,Y 361.889,Z 555.405,A -85,B 0,C 180,E1 -13207.144,E2 -13207.144} C_VEL
LIN {X 0,Y 361.905,Z 555.407,A -85,B 0,C 180,E1 -13210.723,E2 -13210.723} C_VEL
LIN {X 0,Y 361.931,Z 555.401,A -85,B 0,C 180,E1 -13213.065,E2 -13213.065} C_VEL
LIN {X 0,Y 361.997,Z 555.392,A -85,B 0,C 180,E1 -13216.527,E2 -13216.527} C_VEL
LIN {X 0,Y 362.03,Z 555.385,A -85,B 0,C 180,E1 -13219.937,E2 -13219.937} C_VEL
LIN {X 0,Y 362.149,Z 555.37,A -85,B 0,C 180,E1 -13222.192,E2 -13222.192} C_VEL
LIN {X 0,Y 362.117,Z 555.375,A -85,B 0,C 180,E1 -13224.431,E2 -13224.431} C_VEL
LIN {X 0,Y 362.281,Z 555.354,A -85,B 0,C 180,E1 -13227.776,E2 -13227.776} C_VEL
LIN {X 0,Y 362.426,Z 555.336,A -85,B 0,C 180,E1 -13229.999,E2 -13229.999} C_VEL
LIN {X 0,Y 362.281,Z 555.354,A -85,B 0,C 180,E1 -13232.223,E2 -13232.223} C_VEL
LIN {X 0,Y 362.167,Z 555.369,A -85,B 0,C 180,E1 -13236.686,E2 -13236.686} C_VEL
LIN {X 0,Y 362.072,Z 555.382,A -85,B 0,C 180,E1 -13238.933,E2 -13238.933} C_VEL
LIN {X 0,Y 361.964,Z 555.393,A -85,B 0,C 180,E1 -13242.331,E2 -13242.331} C_VEL
LIN {X 0,Y 361.959,Z 555.394,A -85,B 0,C 180,E1 -13244.62,E2 -13244.62} C_VEL
LIN {X 0,Y 361.952,Z 555.396,A -85,B 0,C 180,E1 -13248.099,E2 -13248.099} C_VEL
LIN {X 0,Y 361.889,Z 555.408,A -85,B 0,C 180,E1 -13251.652,E2 -13251.652} C_VEL
LIN {X 0,Y 361.924,Z 555.401,A -85,B 0,C 180,E1 -13255.29,E2 -13255.29} C_VEL
LIN {X 0,Y 361.919,Z 555.404,A -85,B 0,C 180,E1 -13257.777,E2 -13257.777} C_VEL
LIN {X 0,Y 361.857,Z 555.412,A -85,B 0,C 180,E1 -13261.627,E2 -13261.627} C_VEL
LIN {X 0,Y 361.87,Z 555.407,A -85,B 0,C 180,E1 -13265.345,E2 -13265.345} C_VEL
LIN {X 0,Y 361.869,Z 555.405,A -85,B 0,C 180,E1 -13269.027,E2 -13269.027} C_VEL
LIN {X 0,Y 361.862,Z 555.409,A -85,B 0,C 180,E1 -13270.167,E2 -13270.167} C_VEL
LIN {X 0,Y 361.181,Z 555.492,A -85,B 0,C 180,E1 -13271.096,E2 -13271.096} C_VEL
LIN {X 0,Y 358.313,Z 555.849,A -85,B 0,C 180,E1 -13272.606,E2 -13272.606} C_VEL
LIN {X 0,Y 355.908,Z 556.153,A -85,B 0,C 180,E1 -13273.828,E2 -13273.828} C_VEL
LIN {X 0,Y 354.902,Z 556.273,A -85,B 0,C 180,E1 -13274.773,E2 -13274.773} C_VEL
LIN {X 0,Y 354.834,Z 556.281,A -85,B 0,C 180,E1 -13275.093,E2 -13275.093} C_VEL
LIN {X 0,Y 354.835,Z 556.281,A -85,B 0,C 180,E1 -13278.818,E2 -13278.818} C_VEL
LIN {X 0,Y 354.808,Z 556.288,A -85,B 0,C 180,E1 -13282.401,E2 -13282.401} C_VEL
LIN {X 0,Y 354.832,Z 556.282,A -85,B 0,C 180,E1 -13283.141,E2 -13283.141} C_VEL
LIN {X 0,Y 360.258,Z 571.125,A -85,B 0,C 180,E1 -13283.817,E2 -13283.817} C_VEL
LIN {X 0,Y 363.428,Z 580.091,A -85,B 0,C 180,E1 -13284.192,E2 -13284.192} C_VEL
LIN {X 0,Y 362.756,Z 616.989,A -85,B 0,C 180,E1 -13285.084,E2 -13285.084} C_VEL
LIN {X 0,Y 362.539,Z 631.326,A -85,B 0,C 180,E1 -13285.64,E2 -13285.64} C_VEL
LIN {X 0,Y 361.992,Z 645.411,A -85,B 0,C 180,E1 -13286.411,E2 -13286.411} C_VEL
LIN {X 0,Y 361.291,Z 658.104,A -85,B 0,C 180,E1 -13287.33,E2 -13287.33} C_VEL
LIN {X 0,Y 360.442,Z 671.145,A -85,B 0,C 180,E1 -13288.53,E2 -13288.53} C_VEL
LIN {X 0,Y 359.402,Z 683.447,A -85,B 0,C 180,E1 -13289.929,E2 -13289.929} C_VEL
LIN {X 0,Y 358.623,Z 693.344,A -85,B 0,C 180,E1 -13291.307,E2 -13291.307} C_VEL
LIN {X 0,Y 357.795,Z 702.5,A -85,B 0,C 180,E1 -13292.827,E2 -13292.827} C_VEL
LIN {X 0,Y 357.083,Z 710.152,A -85,B 0,C 180,E1 -13294.343,E2 -13294.343} C_VEL
LIN {X 0,Y 356.369,Z 717.794,A -85,B 0,C 180,E1 -13296.154,E2 -13296.154} C_VEL
LIN {X 0,Y 355.743,Z 724.721,A -85,B 0,C 180,E1 -13298.204,E2 -13298.204} C_VEL
LIN {X 0,Y 355.286,Z 730.363,A -85,B 0,C 180,E1 -13300.35,E2 -13300.35} C_VEL
LIN {X 0,Y 355.074,Z 733.398,A -85,B 0,C 180,E1 -13301.815,E2 -13301.815} C_VEL
LIN {X 0,Y 354.821,Z 736.577,A -85,B 0,C 180,E1 -13303.901,E2 -13303.901} C_VEL
LIN {X 0,Y 354.865,Z 738.671,A -85,B 0,C 180,E1 -13306.252,E2 -13306.252} C_VEL
LIN {X 0,Y 355.035,Z 739.299,A -85,B 0,C 180,E1 -13308.583,E2 -13308.583} C_VEL
LIN {X 0,Y 355.348,Z 738.479,A -85,B 0,C 180,E1 -13310.897,E2 -13310.897} C_VEL
LIN {X 0,Y 355.863,Z 736.152,A -85,B 0,C 180,E1 -13313.195,E2 -13313.195} C_VEL
LIN {X 0,Y 356.689,Z 732.31,A -85,B 0,C 180,E1 -13315.48,E2 -13315.48} C_VEL
LIN {X 0,Y 357.353,Z 728.381,A -85,B 0,C 180,E1 -13317.182,E2 -13317.182} C_VEL
LIN {X 0,Y 358.452,Z 722.143,A -85,B 0,C 180,E1 -13319.269,E2 -13319.269} C_VEL
LIN {X 0,Y 359.528,Z 715.163,A -85,B 0,C 180,E1 -13321.121,E2 -13321.121} C_VEL
LIN {X 0,Y 360.817,Z 707.31,A -85,B 0,C 180,E1 -13322.792,E2 -13322.792} C_VEL
LIN {X 0,Y 362.109,Z 697.777,A -85,B 0,C 180,E1 -13324.453,E2 -13324.453} C_VEL
LIN {X 0,Y 363.419,Z 687.084,A -85,B 0,C 180,E1 -13325.967,E2 -13325.967} C_VEL
LIN {X 0,Y 364.732,Z 675.075,A -85,B 0,C 180,E1 -13327.335,E2 -13327.335} C_VEL
LIN {X 0,Y 365.845,Z 663.018,A -85,B 0,C 180,E1 -13328.423,E2 -13328.423} C_VEL
LIN {X 0,Y 366.619,Z 649.703,A -85,B 0,C 180,E1 -13329.378,E2 -13329.378} C_VEL
LIN {X 0,Y 367.171,Z 636.347,A -85,B 0,C 180,E1 -13330.091,E2 -13330.091} C_VEL
LIN {X 0,Y 367.364,Z 622.437,A -85,B 0,C 180,E1 -13330.605,E2 -13330.605} C_VEL
LIN {X 0,Y 367.872,Z 592.133,A -85,B 0,C 180,E1 -13331.36,E2 -13331.36} C_VEL
LIN {X 0,Y 368.101,Z 582.059,A -85,B 0,C 180,E1 -13331.607,E2 -13331.607} C_VEL
LIN {X 0,Y 362.033,Z 569.64,A -85,B 0,C 180,E1 -13332.584,E2 -13332.584} C_VEL
LIN {X 0,Y 356.687,Z 560.105,A -85,B 0,C 180,E1 -13333.475,E2 -13333.475} C_VEL
LIN {X 0,Y 355.201,Z 557.412,A -85,B 0,C 180,E1 -13333.736,E2 -13333.736} C_VEL
LIN {X 0,Y 354.949,Z 556.276,A -85,B 0,C 180,E1 -13333.832,E2 -13333.832} C_VEL
LIN {X 0,Y 354.92,Z 556.277,A -85,B 0,C 180,E1 -13338.109,E2 -13338.109} C_VEL
LIN {X 0,Y 354.832,Z 556.287,A -85,B 0,C 180,E1 -13342.107,E2 -13342.107} C_VEL
LIN {X 0,Y 354.897,Z 556.274,A -85,B 0,C 180,E1 -13345.828,E2 -13345.828} C_VEL
LIN {X 0,Y 354.852,Z 556.275,A -85,B 0,C 180,E1 -13349.679,E2 -13349.679} C_VEL
LIN {X 0,Y 354.804,Z 556.282,A -85,B 0,C 180,E1 -13353.703,E2 -13353.703} C_VEL
LIN {X 0,Y 354.797,Z 556.284,A -85,B 0,C 180,E1 -13356.46,E2 -13356.46} C_VEL
LIN {X 0,Y 354.822,Z 556.282,A -85,B 0,C 180,E1 -13359.424,E2 -13359.424} C_VEL
LIN {X 0,Y 354.787,Z 556.289,A -85,B 0,C 180,E1 -13362.868,E2 -13362.868} C_VEL
LIN {X 0,Y 354.78,Z 556.289,A -85,B 0,C 180,E1 -13366.107,E2 -13366.107} C_VEL
LIN {X 0,Y 354.787,Z 556.283,A -85,B 0,C 180,E1 -13369.18,E2 -13369.18} C_VEL
LIN {X 0,Y 354.895,Z 556.371,A -85,B 0,C 180,E1 -13371.271,E2 -13371.271} C_VEL
LIN {X 0,Y 358.139,Z 572.244,A -85,B 0,C 180,E1 -13375.508,E2 -13375.508} C_VEL
LIN {X 0,Y 359.738,Z 580.145,A -85,B 0,C 180,E1 -13377.534,E2 -13377.534} C_VEL
LIN {X 0,Y 358.081,Z 595.854,A -85,B 0,C 180,E1 -13381.259,E2 -13381.259} C_VEL
LIN {X 0,Y 356.603,Z 612.374,A -85,B 0,C 180,E1 -13385.138,E2 -13385.138} C_VEL
LIN {X 0,Y 356.561,Z 613.153,A -85,B 0,C 180,E1 -13385.282,E2 -13385.282} C_VEL
LIN {X 0,Y 357.3,Z 617.682,A -85,B 0,C 180,E1 -13385.515,E2 -13385.515} C_VEL
LIN {X 0,Y 360.581,Z 637.547,A -85,B 0,C 180,E1 -13386.497,E2 -13386.497} C_VEL
LIN {X 0,Y 364.699,Z 679.926,A -85,B 0,C 180,E1 -13388.188,E2 -13388.188} C_VEL
LIN {X 0,Y 362.931,Z 727.712,A -85,B 0,C 180,E1 -13389.48,E2 -13389.48} C_VEL
LIN {X 0,Y 361.988,Z 741.892,A -85,B 0,C 180,E1 -13390.064,E2 -13390.064} C_VEL
LIN {X 0,Y 360.801,Z 754.919,A -85,B 0,C 180,E1 -13390.811,E2 -13390.811} C_VEL
LIN {X 0,Y 359.335,Z 767.663,A -85,B 0,C 180,E1 -13391.765,E2 -13391.765} C_VEL
LIN {X 0,Y 357.953,Z 779.356,A -85,B 0,C 180,E1 -13392.873,E2 -13392.873} C_VEL
LIN {X 0,Y 356.747,Z 790.09,A -85,B 0,C 180,E1 -13394.138,E2 -13394.138} C_VEL
LIN {X 0,Y 355.599,Z 801.063,A -85,B 0,C 180,E1 -13395.721,E2 -13395.721} C_VEL
LIN {X 0,Y 354.818,Z 810.579,A -85,B 0,C 180,E1 -13397.416,E2 -13397.416} C_VEL
LIN {X 0,Y 354.252,Z 818.403,A -85,B 0,C 180,E1 -13399.137,E2 -13399.137} C_VEL
LIN {X 0,Y 354.073,Z 826.977,A -85,B 0,C 180,E1 -13401.439,E2 -13401.439} C_VEL
LIN {X 0,Y 354.051,Z 832.149,A -85,B 0,C 180,E1 -13403.16,E2 -13403.16} C_VEL
LIN {X 0,Y 354.281,Z 836.123,A -85,B 0,C 180,E1 -13404.879,E2 -13404.879} C_VEL
LIN {X 0,Y 354.34,Z 838.921,A -85,B 0,C 180,E1 -13406.589,E2 -13406.589} C_VEL
LIN {X 0,Y 354.374,Z 840.15,A -85,B 0,C 180,E1 -13407.727,E2 -13407.727} C_VEL
LIN {X 0,Y 354.496,Z 840.942,A -85,B 0,C 180,E1 -13408.865,E2 -13408.865} C_VEL
LIN {X 0,Y 354.695,Z 841.296,A -85,B 0,C 180,E1 -13410.001,E2 -13410.001} C_VEL
LIN {X 0,Y 354.393,Z 841.103,A -85,B 0,C 180,E1 -13411.137,E2 -13411.137} C_VEL
LIN {X 0,Y 354.318,Z 840.46,A -85,B 0,C 180,E1 -13412.274,E2 -13412.274} C_VEL
LIN {X 0,Y 354.272,Z 839.371,A -85,B 0,C 180,E1 -13413.413,E2 -13413.413} C_VEL
LIN {X 0,Y 354.124,Z 836.875,A -85,B 0,C 180,E1 -13415.124,E2 -13415.124} C_VEL
LIN {X 0,Y 353.967,Z 833.161,A -85,B 0,C 180,E1 -13416.9,E2 -13416.9} C_VEL
LIN {X 0,Y 353.919,Z 828.61,A -85,B 0,C 180,E1 -13418.566,E2 -13418.566} C_VEL
LIN {X 0,Y 354.081,Z 821.573,A -85,B 0,C 180,E1 -13420.58,E2 -13420.58} C_VEL
LIN {X 0,Y 354.624,Z 814.102,A -85,B 0,C 180,E1 -13422.302,E2 -13422.302} C_VEL
LIN {X 0,Y 355.24,Z 804.888,A -85,B 0,C 180,E1 -13424.048,E2 -13424.048} C_VEL
LIN {X 0,Y 356.481,Z 794.972,A -85,B 0,C 180,E1 -13425.583,E2 -13425.583} C_VEL
LIN {X 0,Y 357.883,Z 784.009,A -85,B 0,C 180,E1 -13426.985,E2 -13426.985} C_VEL
LIN {X 0,Y 359.451,Z 772.192,A -85,B 0,C 180,E1 -13428.231,E2 -13428.231} C_VEL
LIN {X 0,Y 361.031,Z 759.415,A -85,B 0,C 180,E1 -13429.326,E2 -13429.326} C_VEL
LIN {X 0,Y 362.893,Z 744.276,A -85,B 0,C 180,E1 -13430.328,E2 -13430.328} C_VEL
LIN {X 0,Y 364.317,Z 729.707,A -85,B 0,C 180,E1 -13431.057,E2 -13431.057} C_VEL
LIN {X 0,Y 365.414,Z 713.298,A -85,B 0,C 180,E1 -13431.641,E2 -13431.641} C_VEL
LIN {X 0,Y 366.858,Z 679.222,A -85,B 0,C 180,E1 -13432.613,E2 -13432.613} C_VEL
LIN {X 0,Y 365.632,Z 646.613,A -85,B 0,C 180,E1 -13433.856,E2 -13433.856} C_VEL
LIN {X 0,Y 363.846,Z 627.603,A -85,B 0,C 180,E1 -13434.744,E2 -13434.744} C_VEL
LIN {X 0,Y 361.191,Z 610.173,A -85,B 0,C 180,E1 -13435.729,E2 -13435.729} C_VEL
LIN {X 0,Y 358.592,Z 596.089,A -85,B 0,C 180,E1 -13436.636,E2 -13436.636} C_VEL
LIN {X 0,Y 356.79,Z 588.282,A -85,B 0,C 180,E1 -13437.217,E2 -13437.217} C_VEL
LIN {X 0,Y 355.929,Z 583.263,A -85,B 0,C 180,E1 -13437.583,E2 -13437.583} C_VEL
LIN {X 0,Y 356.785,Z 569.321,A -85,B 0,C 180,E1 -13440.808,E2 -13440.808} C_VEL
LIN {X 0,Y 356.466,Z 564.347,A -85,B 0,C 180,E1 -13442.028,E2 -13442.028} C_VEL
LIN {X 0,Y 354.909,Z 556.279,A -85,B 0,C 180,E1 -13444.187,E2 -13444.187} C_VEL
LIN {X 0,Y 354.81,Z 556.286,A -85,B 0,C 180,E1 -13447.883,E2 -13447.883} C_VEL
LIN {X 0,Y 354.792,Z 556.291,A -85,B 0,C 180,E1 -13451.172,E2 -13451.172} C_VEL
LIN {X 0,Y 354.768,Z 556.291,A -85,B 0,C 180,E1 -13454.506,E2 -13454.506} C_VEL
LIN {X 0,Y 354.799,Z 556.29,A -85,B 0,C 180,E1 -13457.663,E2 -13457.663} C_VEL
LIN {X 0,Y 354.82,Z 556.285,A -85,B 0,C 180,E1 -13460.666,E2 -13460.666} C_VEL
LIN {X 0,Y 354.826,Z 556.285,A -85,B 0,C 180,E1 -13464.301,E2 -13464.301} C_VEL
LIN {X 0,Y 354.791,Z 556.29,A -85,B 0,C 180,E1 -13467.667,E2 -13467.667} C_VEL
LIN {X 0,Y 354.851,Z 556.285,A -85,B 0,C 180,E1 -13471.619,E2 -13471.619} C_VEL
LIN {X 0,Y 354.896,Z 556.349,A -85,B 0,C 180,E1 -13472.617,E2 -13472.617} C_VEL
LIN {X 0,Y 355.865,Z 559.085,A -85,B 0,C 180,E1 -13472.871,E2 -13472.871} C_VEL
LIN {X 0,Y 357.802,Z 561.519,A -85,B 0,C 180,E1 -13473.258,E2 -13473.258} C_VEL
LIN {X 0,Y 364.21,Z 572.058,A -85,B 0,C 180,E1 -13474.491,E2 -13474.491} C_VEL
LIN {X 0,Y 369.684,Z 582.5,A -85,B 0,C 180,E1 -13475.469,E2 -13475.469} C_VEL
LIN {X 0,Y 371.074,Z 585.895,A -85,B 0,C 180,E1 -13475.73,E2 -13475.73} C_VEL
LIN {X 0,Y 370.68,Z 612.786,A -85,B 0,C 180,E1 -13476.422,E2 -13476.422} C_VEL
LIN {X 0,Y 370.534,Z 627.181,A -85,B 0,C 180,E1 -13476.965,E2 -13476.965} C_VEL
LIN {X 0,Y 369.963,Z 641.83,A -85,B 0,C 180,E1 -13477.744,E2 -13477.744} C_VEL
LIN {X 0,Y 368.99,Z 656.536,A -85,B 0,C 180,E1 -13478.783,E2 -13478.783} C_VEL
LIN {X 0,Y 367.879,Z 668.887,A -85,B 0,C 180,E1 -13479.886,E2 -13479.886} C_VEL
LIN {X 0,Y 366.474,Z 681.32,A -85,B 0,C 180,E1 -13481.263,E2 -13481.263} C_VEL
LIN {X 0,Y 365.087,Z 691.578,A -85,B 0,C 180,E1 -13482.639,E2 -13482.639} C_VEL
LIN {X 0,Y 363.484,Z 701.859,A -85,B 0,C 180,E1 -13484.294,E2 -13484.294} C_VEL
LIN {X 0,Y 362.053,Z 710.43,A -85,B 0,C 180,E1 -13485.957,E2 -13485.957} C_VEL
LIN {X 0,Y 360.534,Z 718.651,A -85,B 0,C 180,E1 -13487.903,E2 -13487.903} C_VEL
LIN {X 0,Y 359.221,Z 725.333,A -85,B 0,C 180,E1 -13489.858,E2 -13489.858} C_VEL
LIN {X 0,Y 357.838,Z 731.425,A -85,B 0,C 180,E1 -13492.097,E2 -13492.097} C_VEL
LIN {X 0,Y 357.228,Z 734.96,A -85,B 0,C 180,E1 -13493.788,E2 -13493.788} C_VEL
LIN {X 0,Y 356.598,Z 737.679,A -85,B 0,C 180,E1 -13495.478,E2 -13495.478} C_VEL
LIN {X 0,Y 355.901,Z 740.201,A -85,B 0,C 180,E1 -13497.736,E2 -13497.736} C_VEL
LIN {X 0,Y 355.471,Z 741.454,A -85,B 0,C 180,E1 -13499.999,E2 -13499.999} C_VEL
LIN {X 0,Y 355.166,Z 741.489,A -85,B 0,C 180,E1 -13502.268,E2 -13502.268} C_VEL
LIN {X 0,Y 354.926,Z 740.299,A -85,B 0,C 180,E1 -13504.542,E2 -13504.542} C_VEL
LIN {X 0,Y 355.235,Z 737.804,A -85,B 0,C 180,E1 -13506.817,E2 -13506.817} C_VEL
LIN {X 0,Y 355.354,Z 734.04,A -85,B 0,C 180,E1 -13509.103,E2 -13509.103} C_VEL
LIN {X 0,Y 355.665,Z 728.863,A -85,B 0,C 180,E1 -13511.396,E2 -13511.396} C_VEL
LIN {X 0,Y 356.192,Z 722.125,A -85,B 0,C 180,E1 -13513.695,E2 -13513.695} C_VEL
LIN {X 0,Y 356.864,Z 714.878,A -85,B 0,C 180,E1 -13515.681,E2 -13515.681} C_VEL
LIN {X 0,Y 357.745,Z 705.788,A -85,B 0,C 180,E1 -13517.728,E2 -13517.728} C_VEL
LIN {X 0,Y 358.673,Z 696.552,A -85,B 0,C 180,E1 -13519.457,E2 -13519.457} C_VEL
LIN {X 0,Y 359.665,Z 685.507,A -85,B 0,C 180,E1 -13521.192,E2 -13521.192} C_VEL
LIN {X 0,Y 360.7,Z 673.311,A -85,B 0,C 180,E1 -13522.783,E2 -13522.783} C_VEL
LIN {X 0,Y 361.652,Z 661.289,A -85,B 0,C 180,E1 -13524.085,E2 -13524.085} C_VEL
LIN {X 0,Y 362.601,Z 648.356,A -85,B 0,C 180,E1 -13525.239,E2 -13525.239} C_VEL
LIN {X 0,Y 363.364,Z 634.219,A -85,B 0,C 180,E1 -13526.259,E2 -13526.259} C_VEL
LIN {X 0,Y 364.021,Z 619.258,A -85,B 0,C 180,E1 -13527.09,E2 -13527.09} C_VEL
LIN {X 0,Y 364.358,Z 603.849,A -85,B 0,C 180,E1 -13527.715,E2 -13527.715} C_VEL
LIN {X 0,Y 364.423,Z 582.122,A -85,B 0,C 180,E1 -13528.304,E2 -13528.304} C_VEL
LIN {X 0,Y 354.844,Z 556.284,A -85,B 0,C 180,E1 -13529.493,E2 -13529.493} C_VEL
LIN {X 0,Y 354.788,Z 556.291,A -85,B 0,C 180,E1 -13532.333,E2 -13532.333} C_VEL
LIN {X 0,Y 354.823,Z 556.285,A -85,B 0,C 180,E1 -13535.699,E2 -13535.699} C_VEL
LIN {X 0,Y 354.825,Z 556.283,A -85,B 0,C 180,E1 -13539.423,E2 -13539.423} C_VEL
LIN {X 0,Y 354.788,Z 556.288,A -85,B 0,C 180,E1 -13542.866,E2 -13542.866} C_VEL
LIN {X 0,Y 354.767,Z 556.294,A -85,B 0,C 180,E1 -13546.103,E2 -13546.103} C_VEL
LIN {X 0,Y 354.788,Z 556.287,A -85,B 0,C 180,E1 -13549.178,E2 -13549.178} C_VEL
LIN {X 0,Y 354.812,Z 556.29,A -85,B 0,C 180,E1 -13552.401,E2 -13552.401} C_VEL
LIN {X 0,Y 354.811,Z 556.286,A -85,B 0,C 180,E1 -13554.94,E2 -13554.94} C_VEL
LIN {X 0,Y 354.793,Z 556.291,A -85,B 0,C 180,E1 -13558.404,E2 -13558.404} C_VEL
LIN {X 0,Y 354.845,Z 556.28,A -85,B 0,C 180,E1 -13561.618,E2 -13561.618} C_VEL
LIN {X 0,Y 354.898,Z 556.275,A -85,B 0,C 180,E1 -13564.172,E2 -13564.172} C_VEL
LIN {X 0,Y 354.834,Z 556.282,A -85,B 0,C 180,E1 -13567.893,E2 -13567.893} C_VEL
LIN {X 0,Y 354.921,Z 556.271,A -85,B 0,C 180,E1 -13571.891,E2 -13571.891} C_VEL
LIN {X 0,Y 354.941,Z 556.268,A -85,B 0,C 180,E1 -13575.98,E2 -13575.98} C_VEL
LIN {X 0,Y 354.976,Z 556.264,A -85,B 0,C 180,E1 -13579.735,E2 -13579.735} C_VEL
LIN {X 0,Y 355.112,Z 556.247,A -85,B 0,C 180,E1 -13582.036,E2 -13582.036} C_VEL
LIN {X 0,Y 355.091,Z 556.25,A -85,B 0,C 180,E1 -13584.32,E2 -13584.32} C_VEL
LIN {X 0,Y 355.244,Z 556.231,A -85,B 0,C 180,E1 -13587.732,E2 -13587.732} C_VEL
LIN {X 0,Y 355.395,Z 556.212,A -85,B 0,C 180,E1 -13589.999,E2 -13589.999} C_VEL
LIN {X 0,Y 355.244,Z 556.23,A -85,B 0,C 180,E1 -13592.267,E2 -13592.267} C_VEL
LIN {X 0,Y 355.133,Z 556.246,A -85,B 0,C 180,E1 -13596.819,E2 -13596.819} C_VEL
LIN {X 0,Y 355.013,Z 556.264,A -85,B 0,C 180,E1 -13599.112,E2 -13599.112} C_VEL
LIN {X 0,Y 354.924,Z 556.271,A -85,B 0,C 180,E1 -13602.58,E2 -13602.58} C_VEL
LIN {X 0,Y 354.886,Z 556.276,A -85,B 0,C 180,E1 -13606.095,E2 -13606.095} C_VEL
LIN {X 0,Y 354.897,Z 556.273,A -85,B 0,C 180,E1 -13608.472,E2 -13608.472} C_VEL
LIN {X 0,Y 354.832,Z 556.283,A -85,B 0,C 180,E1 -13612.105,E2 -13612.105} C_VEL
LIN {X 0,Y 354.895,Z 556.278,A -85,B 0,C 180,E1 -13615.827,E2 -13615.827} C_VEL
LIN {X 0,Y 354.85,Z 556.286,A -85,B 0,C 180,E1 -13619.678,E2 -13619.678} C_VEL
LIN {X 0,Y 354.825,Z 556.288,A -85,B 0,C 180,E1 -13623.682,E2 -13623.682} C_VEL
LIN {X 0,Y 354.797,Z 556.287,A -85,B 0,C 180,E1 -13626.459,E2 -13626.459} C_VEL
LIN {X 0,Y 354.793,Z 556.284,A -85,B 0,C 180,E1 -13630.168,E2 -13630.168} C_VEL
LIN {X 0,Y 354.8,Z 556.292,A -85,B 0,C 180,E1 -13633.89,E2 -13633.89} C_VEL
LIN {X 0,Y 354.834,Z 556.281,A -85,B 0,C 180,E1 -13635.093,E2 -13635.093} C_VEL
LIN {X 0,Y 354.199,Z 556.367,A -85,B 0,C 180,E1 -13636.041,E2 -13636.041} C_VEL
LIN {X 0,Y 351.343,Z 556.718,A -85,B 0,C 180,E1 -13637.582,E2 -13637.582} C_VEL
LIN {X 0,Y 348.905,Z 557.021,A -85,B 0,C 180,E1 -13638.83,E2 -13638.83} C_VEL
LIN {X 0,Y 347.862,Z 557.154,A -85,B 0,C 180,E1 -13639.796,E2 -13639.796} C_VEL
LIN {X 0,Y 347.78,Z 557.165,A -85,B 0,C 180,E1 -13640.123,E2 -13640.123} C_VEL
LIN {X 0,Y 347.789,Z 557.16,A -85,B 0,C 180,E1 -13642.78,E2 -13642.78} C_VEL
LIN {X 0,Y 352.402,Z 569.789,A -85,B 0,C 180,E1 -13643.38,E2 -13643.38} C_VEL
LIN {X 0,Y 356.581,Z 581.008,A -85,B 0,C 180,E1 -13643.875,E2 -13643.875} C_VEL
LIN {X 0,Y 355.886,Z 619.484,A -85,B 0,C 180,E1 -13644.84,E2 -13644.84} C_VEL
LIN {X 0,Y 355.687,Z 632.869,A -85,B 0,C 180,E1 -13645.385,E2 -13645.385} C_VEL
LIN {X 0,Y 355.122,Z 646.928,A -85,B 0,C 180,E1 -13646.18,E2 -13646.18} C_VEL
LIN {X 0,Y 354.395,Z 659.567,A -85,B 0,C 180,E1 -13647.121,E2 -13647.121} C_VEL
LIN {X 0,Y 353.488,Z 672.836,A -85,B 0,C 180,E1 -13648.374,E2 -13648.374} C_VEL
LIN {X 0,Y 352.439,Z 684.788,A -85,B 0,C 180,E1 -13649.768,E2 -13649.768} C_VEL
LIN {X 0,Y 351.555,Z 695.625,A -85,B 0,C 180,E1 -13651.329,E2 -13651.329} C_VEL
LIN {X 0,Y 350.673,Z 704.568,A -85,B 0,C 180,E1 -13652.875,E2 -13652.875} C_VEL
LIN {X 0,Y 349.924,Z 713.107,A -85,B 0,C 180,E1 -13654.66,E2 -13654.66} C_VEL
LIN {X 0,Y 349.194,Z 720.644,A -85,B 0,C 180,E1 -13656.579,E2 -13656.579} C_VEL
LIN {X 0,Y 348.596,Z 727.379,A -85,B 0,C 180,E1 -13658.722,E2 -13658.722} C_VEL
LIN {X 0,Y 348.219,Z 731.868,A -85,B 0,C 180,E1 -13660.549,E2 -13660.549} C_VEL
LIN {X 0,Y 347.945,Z 735.33,A -85,B 0,C 180,E1 -13662.364,E2 -13662.364} C_VEL
LIN {X 0,Y 347.793,Z 738.531,A -85,B 0,C 180,E1 -13664.77,E2 -13664.77} C_VEL
LIN {X 0,Y 347.826,Z 739.528,A -85,B 0,C 180,E1 -13665.968,E2 -13665.968} C_VEL
LIN {X 0,Y 347.984,Z 740.382,A -85,B 0,C 180,E1 -13668.349,E2 -13668.349} C_VEL
LIN {X 0,Y 348.335,Z 739.787,A -85,B 0,C 180,E1 -13670.712,E2 -13670.712} C_VEL
LIN {X 0,Y 348.853,Z 737.755,A -85,B 0,C 180,E1 -13673.058,E2 -13673.058} C_VEL
LIN {X 0,Y 349.708,Z 734.128,A -85,B 0,C 180,E1 -13675.39,E2 -13675.39} C_VEL
LIN {X 0,Y 350.689,Z 728.969,A -85,B 0,C 180,E1 -13677.703,E2 -13677.703} C_VEL
LIN {X 0,Y 351.879,Z 722.677,A -85,B 0,C 180,E1 -13679.808,E2 -13679.808} C_VEL
LIN {X 0,Y 353.052,Z 715.42,A -85,B 0,C 180,E1 -13681.712,E2 -13681.712} C_VEL
LIN {X 0,Y 354.456,Z 707.334,A -85,B 0,C 180,E1 -13683.411,E2 -13683.411} C_VEL
LIN {X 0,Y 355.81,Z 697.575,A -85,B 0,C 180,E1 -13685.1,E2 -13685.1} C_VEL
LIN {X 0,Y 357.143,Z 687.704,A -85,B 0,C 180,E1 -13686.497,E2 -13686.497} C_VEL
LIN {X 0,Y 358.372,Z 676.956,A -85,B 0,C 180,E1 -13687.749,E2 -13687.749} C_VEL
LIN {X 0,Y 359.556,Z 665.081,A -85,B 0,C 180,E1 -13688.855,E2 -13688.855} C_VEL
LIN {X 0,Y 360.394,Z 651.938,A -85,B 0,C 180,E1 -13689.825,E2 -13689.825} C_VEL
LIN {X 0,Y 360.995,Z 638.238,A -85,B 0,C 180,E1 -13690.581,E2 -13690.581} C_VEL
LIN {X 0,Y 361.221,Z 624.324,A -85,B 0,C 180,E1 -13691.12,E2 -13691.12} C_VEL
LIN {X 0,Y 361.881,Z 591.899,A -85,B 0,C 180,E1 -13691.958,E2 -13691.958} C_VEL
LIN {X 0,Y 362.054,Z 584.244,A -85,B 0,C 180,E1 -13692.159,E2 -13692.159} C_VEL
LIN {X 0,Y 355.718,Z 571.469,A -85,B 0,C 180,E1 -13693.231,E2 -13693.231} C_VEL
LIN {X 0,Y 351.511,Z 564.144,A -85,B 0,C 180,E1 -13693.964,E2 -13693.964} C_VEL
LIN {X 0,Y 349.701,Z 561.066,A -85,B 0,C 180,E1 -13694.292,E2 -13694.292} C_VEL
LIN {X 0,Y 348.174,Z 558.483,A -85,B 0,C 180,E1 -13694.579,E2 -13694.579} C_VEL
LIN {X 0,Y 347.892,Z 557.155,A -85,B 0,C 180,E1 -13694.687,E2 -13694.687} C_VEL
LIN {X 0,Y 347.853,Z 557.159,A -85,B 0,C 180,E1 -13698.861,E2 -13698.861} C_VEL
LIN {X 0,Y 347.771,Z 557.166,A -85,B 0,C 180,E1 -13702.58,E2 -13702.58} C_VEL
LIN {X 0,Y 347.81,Z 557.158,A -85,B 0,C 180,E1 -13705.109,E2 -13705.109} C_VEL
LIN {X 0,Y 347.81,Z 557.154,A -85,B 0,C 180,E1 -13707.694,E2 -13707.694} C_VEL
LIN {X 0,Y 347.762,Z 557.157,A -85,B 0,C 180,E1 -13710.347,E2 -13710.347} C_VEL
LIN {X 0,Y 347.742,Z 557.159,A -85,B 0,C 180,E1 -13714.465,E2 -13714.465} C_VEL
LIN {X 0,Y 347.773,Z 557.162,A -85,B 0,C 180,E1 -13717.99,E2 -13717.99} C_VEL
LIN {X 0,Y 347.75,Z 557.163,A -85,B 0,C 180,E1 -13721.831,E2 -13721.831} C_VEL
LIN {X 0,Y 347.765,Z 557.167,A -85,B 0,C 180,E1 -13725.018,E2 -13725.018} C_VEL
LIN {X 0,Y 347.749,Z 557.16,A -85,B 0,C 180,E1 -13728.398,E2 -13728.398} C_VEL
LIN {X 0,Y 347.829,Z 557.215,A -85,B 0,C 180,E1 -13731.033,E2 -13731.033} C_VEL
LIN {X 0,Y 350.921,Z 572.495,A -85,B 0,C 180,E1 -13735.198,E2 -13735.198} C_VEL
LIN {X 0,Y 352.715,Z 581.102,A -85,B 0,C 180,E1 -13737.454,E2 -13737.454} C_VEL
LIN {X 0,Y 350.993,Z 596.873,A -85,B 0,C 180,E1 -13741.279,E2 -13741.279} C_VEL
LIN {X 0,Y 349.793,Z 609.835,A -85,B 0,C 180,E1 -13744.391,E2 -13744.391} C_VEL
LIN {X 0,Y 350.595,Z 614.912,A -85,B 0,C 180,E1 -13744.677,E2 -13744.677} C_VEL
